// TIA Portal V17 export
// export: Created 2025-03-07T09:19:12.1414983Z, ExportSetting WithDefaults, DisplayName Totally Integrated Automation Portal, DisplayVersion V17 Update 8, DisplayName TIA Portal Openness, DisplayVersion V17 Update 8, DisplayName TIA Portal Version Control Interface, DisplayVersion V17, DisplayName SINAMICS Startdrive Advanced, DisplayVersion V17 SP2, DisplayName SINAMICS Startdrive G110M, G120, G120C, G120D, G120P, G115D, DisplayVersion V17 SP2, DisplayName SINAMICS Startdrive G130, G150, S120, S150, SINAMICS MV, S210, DisplayVersion V17 SP2, DisplayName STEP 7 Professional, DisplayVersion V17 Update 8, DisplayName SINUMERIK ONE STEP 7 Toolbox, DisplayVersion V17 Update 12, DisplayName SINUMERIK 840D sl STEP 7 Toolbox, DisplayVersion V17 Update 12, DisplayName STEP 7 Safety, DisplayVersion V17 Update 6, DisplayName WinCC Advanced, DisplayVersion V17 Update 8
FUNCTION "FC7225_HMI_AXES_CLADDING" : Void   // FC7225, LAD
{ S7_Optimized_Access := 'FALSE' }
AUTHOR : ETXETAR
VERSION : 1.0
// stored: AutoNumber false, IsIECCheckEnabled false, SetENOAutomatically false, UDAEnableTagReadback false
   VAR_TEMP
      ZERO : Byte;
      SOFTKEY_SELECT_PLUS : Byte;   // SOFTKEY_SELECT_PLUS
      SOFTKEY_SELECT_MINUS : Byte;   // SOFTKEY_SELECT_MINUS
      AXIS_SCREEN_SELECTED : Bool;   // AXIS SCREEN SELECTED
      SELECTED_AXIS : Int;   // SELECTED AXIS
   END_VAR
   VAR_TEMP   // added for the SCL form of the ladder/FBD networks
      _w1 : Bool;
      _w2 : Bool;
      _w3 : Bool;
      _w4 : Bool;
   END_VAR
BEGIN

REGION Network 1: ZERO
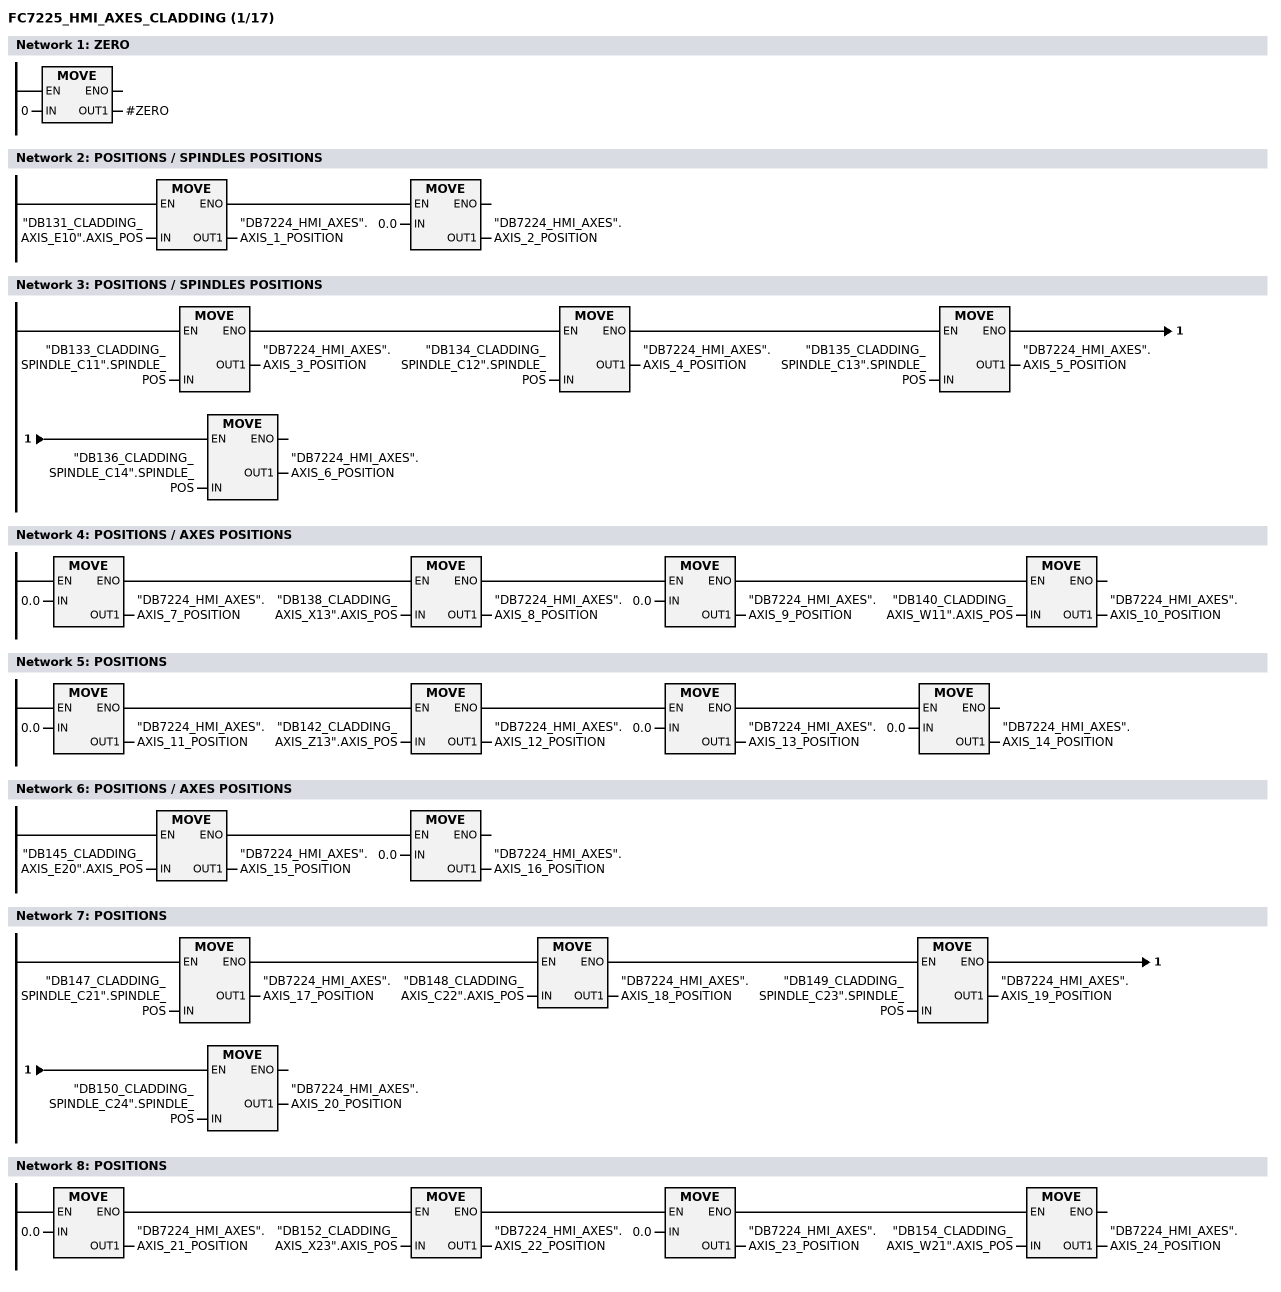
   RUNG wire#powerrail
      { S7_GenerateENO := "TRUE" } Move(in := 0, out1 => #ZERO)
   END_RUNG
   // the same network as SCL:
   #ZERO := 0;
END_REGION

REGION Network 2: POSITIONS / SPINDLES POSITIONS
   RUNG wire#powerrail
      { S7_GenerateENO := "TRUE" } Move(in := "DB131_CLADDING_AXIS_E10".AXIS_POS, out1 => "DB7224_HMI_AXES".AXIS_1_POSITION)
      { S7_GenerateENO := "TRUE" } Move(in := 0.0, out1 => "DB7224_HMI_AXES".AXIS_2_POSITION)
   END_RUNG
   // the same network as SCL:
   // ENO of a box is taken as its EN; it also drops when the box reports an error
   "DB7224_HMI_AXES".AXIS_1_POSITION := "DB131_CLADDING_AXIS_E10".AXIS_POS;
   "DB7224_HMI_AXES".AXIS_2_POSITION := 0.0;
END_REGION

REGION Network 3: POSITIONS / SPINDLES POSITIONS
   RUNG wire#powerrail
      { S7_GenerateENO := "TRUE" } Move(in := "DB133_CLADDING_SPINDLE_C11".SPINDLE_POS, out1 => "DB7224_HMI_AXES".AXIS_3_POSITION)
      { S7_GenerateENO := "TRUE" } Move(in := "DB134_CLADDING_SPINDLE_C12".SPINDLE_POS, out1 => "DB7224_HMI_AXES".AXIS_4_POSITION)
      { S7_GenerateENO := "TRUE" } Move(in := "DB135_CLADDING_SPINDLE_C13".SPINDLE_POS, out1 => "DB7224_HMI_AXES".AXIS_5_POSITION)
      { S7_GenerateENO := "TRUE" } Move(in := "DB136_CLADDING_SPINDLE_C14".SPINDLE_POS, out1 => "DB7224_HMI_AXES".AXIS_6_POSITION)
   END_RUNG
   // the same network as SCL:
   // ENO of a box is taken as its EN; it also drops when the box reports an error
   "DB7224_HMI_AXES".AXIS_3_POSITION := "DB133_CLADDING_SPINDLE_C11".SPINDLE_POS;
   "DB7224_HMI_AXES".AXIS_4_POSITION := "DB134_CLADDING_SPINDLE_C12".SPINDLE_POS;
   "DB7224_HMI_AXES".AXIS_5_POSITION := "DB135_CLADDING_SPINDLE_C13".SPINDLE_POS;
   "DB7224_HMI_AXES".AXIS_6_POSITION := "DB136_CLADDING_SPINDLE_C14".SPINDLE_POS;
END_REGION

REGION Network 4: POSITIONS / AXES POSITIONS
   RUNG wire#powerrail
      { S7_GenerateENO := "TRUE" } Move(in := 0.0, out1 => "DB7224_HMI_AXES".AXIS_7_POSITION)
      { S7_GenerateENO := "TRUE" } Move(in := "DB138_CLADDING_AXIS_X13".AXIS_POS, out1 => "DB7224_HMI_AXES".AXIS_8_POSITION)
      { S7_GenerateENO := "TRUE" } Move(in := 0.0, out1 => "DB7224_HMI_AXES".AXIS_9_POSITION)
      { S7_GenerateENO := "TRUE" } Move(in := "DB140_CLADDING_AXIS_W11".AXIS_POS, out1 => "DB7224_HMI_AXES".AXIS_10_POSITION)
   END_RUNG
   // the same network as SCL:
   // ENO of a box is taken as its EN; it also drops when the box reports an error
   "DB7224_HMI_AXES".AXIS_7_POSITION := 0.0;
   "DB7224_HMI_AXES".AXIS_8_POSITION := "DB138_CLADDING_AXIS_X13".AXIS_POS;
   "DB7224_HMI_AXES".AXIS_9_POSITION := 0.0;
   "DB7224_HMI_AXES".AXIS_10_POSITION := "DB140_CLADDING_AXIS_W11".AXIS_POS;
END_REGION

REGION Network 5: POSITIONS
   RUNG wire#powerrail
      { S7_GenerateENO := "TRUE" } Move(in := 0.0, out1 => "DB7224_HMI_AXES".AXIS_11_POSITION)
      { S7_GenerateENO := "TRUE" } Move(in := "DB142_CLADDING_AXIS_Z13".AXIS_POS, out1 => "DB7224_HMI_AXES".AXIS_12_POSITION)
      { S7_GenerateENO := "TRUE" } Move(in := 0.0, out1 => "DB7224_HMI_AXES".AXIS_13_POSITION)
      { S7_GenerateENO := "TRUE" } Move(in := 0.0, out1 => "DB7224_HMI_AXES".AXIS_14_POSITION)
   END_RUNG
   // the same network as SCL:
   // ENO of a box is taken as its EN; it also drops when the box reports an error
   "DB7224_HMI_AXES".AXIS_11_POSITION := 0.0;
   "DB7224_HMI_AXES".AXIS_12_POSITION := "DB142_CLADDING_AXIS_Z13".AXIS_POS;
   "DB7224_HMI_AXES".AXIS_13_POSITION := 0.0;
   "DB7224_HMI_AXES".AXIS_14_POSITION := 0.0;
END_REGION

REGION Network 6: POSITIONS / AXES POSITIONS
   RUNG wire#powerrail
      { S7_GenerateENO := "TRUE" } Move(in := "DB145_CLADDING_AXIS_E20".AXIS_POS, out1 => "DB7224_HMI_AXES".AXIS_15_POSITION)
      { S7_GenerateENO := "TRUE" } Move(in := 0.0, out1 => "DB7224_HMI_AXES".AXIS_16_POSITION)
   END_RUNG
   // the same network as SCL:
   // ENO of a box is taken as its EN; it also drops when the box reports an error
   "DB7224_HMI_AXES".AXIS_15_POSITION := "DB145_CLADDING_AXIS_E20".AXIS_POS;
   "DB7224_HMI_AXES".AXIS_16_POSITION := 0.0;
END_REGION

REGION Network 7: POSITIONS
   RUNG wire#powerrail
      { S7_GenerateENO := "TRUE" } Move(in := "DB147_CLADDING_SPINDLE_C21".SPINDLE_POS, out1 => "DB7224_HMI_AXES".AXIS_17_POSITION)
      { S7_GenerateENO := "TRUE" } Move(in := "DB148_CLADDING_AXIS_C22".AXIS_POS, out1 => "DB7224_HMI_AXES".AXIS_18_POSITION)
      { S7_GenerateENO := "TRUE" } Move(in := "DB149_CLADDING_SPINDLE_C23".SPINDLE_POS, out1 => "DB7224_HMI_AXES".AXIS_19_POSITION)
      { S7_GenerateENO := "TRUE" } Move(in := "DB150_CLADDING_SPINDLE_C24".SPINDLE_POS, out1 => "DB7224_HMI_AXES".AXIS_20_POSITION)
   END_RUNG
   // the same network as SCL:
   // ENO of a box is taken as its EN; it also drops when the box reports an error
   "DB7224_HMI_AXES".AXIS_17_POSITION := "DB147_CLADDING_SPINDLE_C21".SPINDLE_POS;
   "DB7224_HMI_AXES".AXIS_18_POSITION := "DB148_CLADDING_AXIS_C22".AXIS_POS;
   "DB7224_HMI_AXES".AXIS_19_POSITION := "DB149_CLADDING_SPINDLE_C23".SPINDLE_POS;
   "DB7224_HMI_AXES".AXIS_20_POSITION := "DB150_CLADDING_SPINDLE_C24".SPINDLE_POS;
END_REGION

REGION Network 8: POSITIONS
   RUNG wire#powerrail
      { S7_GenerateENO := "TRUE" } Move(in := 0.0, out1 => "DB7224_HMI_AXES".AXIS_21_POSITION)
      { S7_GenerateENO := "TRUE" } Move(in := "DB152_CLADDING_AXIS_X23".AXIS_POS, out1 => "DB7224_HMI_AXES".AXIS_22_POSITION)
      { S7_GenerateENO := "TRUE" } Move(in := 0.0, out1 => "DB7224_HMI_AXES".AXIS_23_POSITION)
      { S7_GenerateENO := "TRUE" } Move(in := "DB154_CLADDING_AXIS_W21".AXIS_POS, out1 => "DB7224_HMI_AXES".AXIS_24_POSITION)
   END_RUNG
   // the same network as SCL:
   // ENO of a box is taken as its EN; it also drops when the box reports an error
   "DB7224_HMI_AXES".AXIS_21_POSITION := 0.0;
   "DB7224_HMI_AXES".AXIS_22_POSITION := "DB152_CLADDING_AXIS_X23".AXIS_POS;
   "DB7224_HMI_AXES".AXIS_23_POSITION := 0.0;
   "DB7224_HMI_AXES".AXIS_24_POSITION := "DB154_CLADDING_AXIS_W21".AXIS_POS;
END_REGION

REGION Network 9: POSITIONS
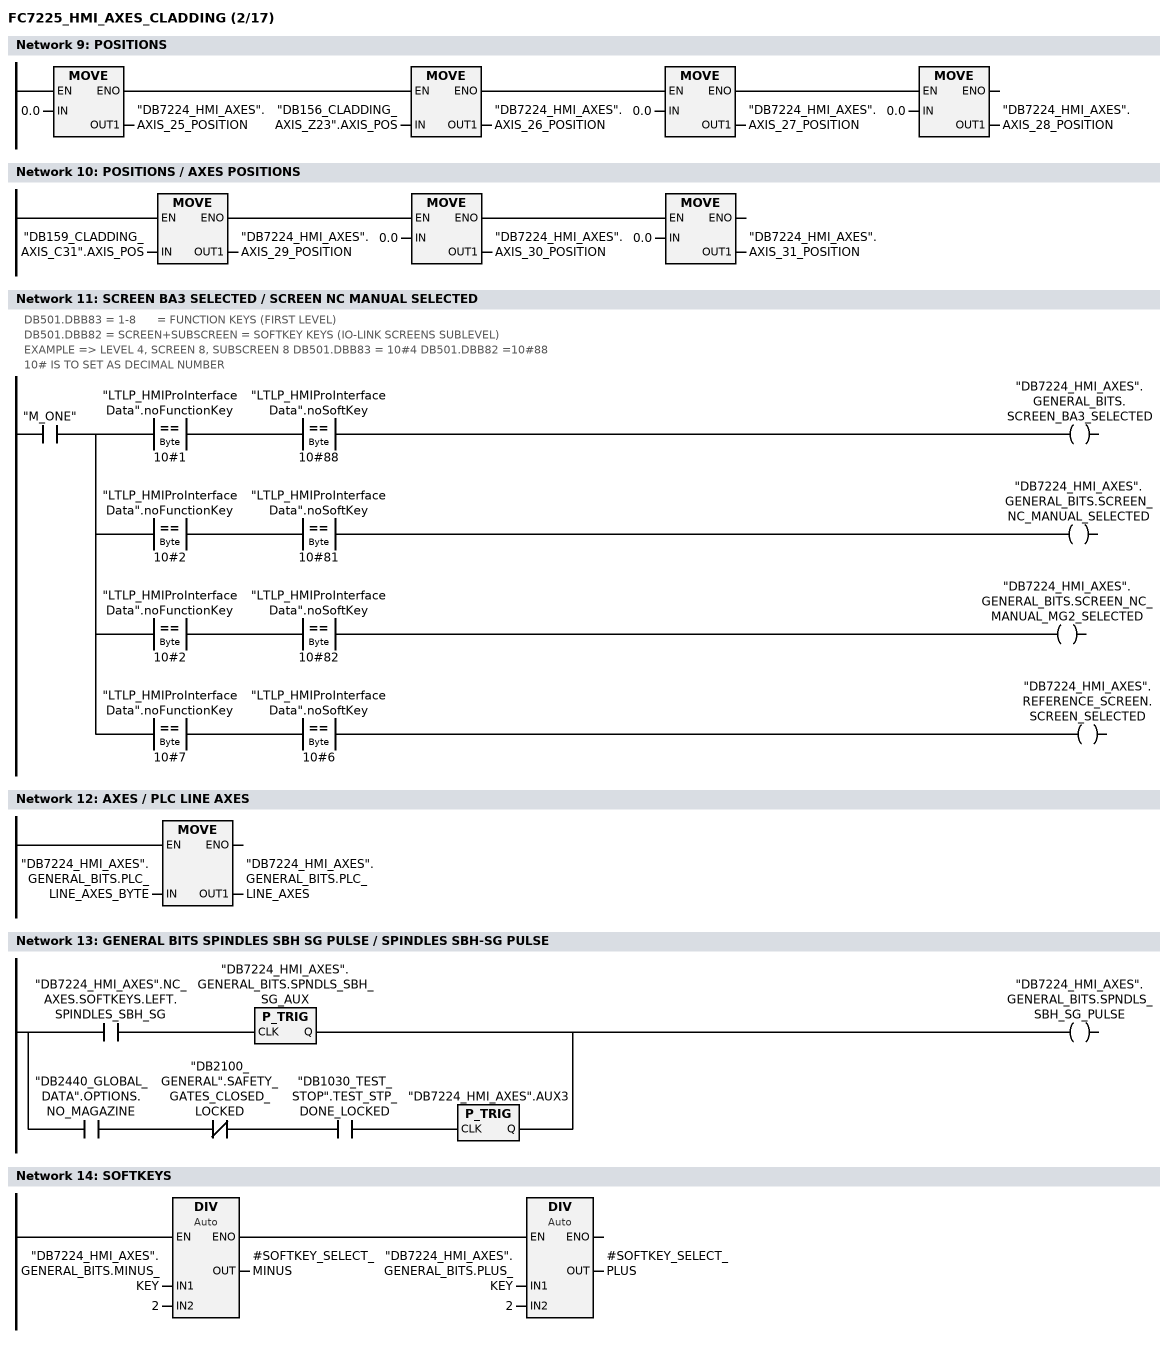
   RUNG wire#powerrail
      { S7_GenerateENO := "TRUE" } Move(in := 0.0, out1 => "DB7224_HMI_AXES".AXIS_25_POSITION)
      { S7_GenerateENO := "TRUE" } Move(in := "DB156_CLADDING_AXIS_Z23".AXIS_POS, out1 => "DB7224_HMI_AXES".AXIS_26_POSITION)
      { S7_GenerateENO := "TRUE" } Move(in := 0.0, out1 => "DB7224_HMI_AXES".AXIS_27_POSITION)
      { S7_GenerateENO := "TRUE" } Move(in := 0.0, out1 => "DB7224_HMI_AXES".AXIS_28_POSITION)
   END_RUNG
   // the same network as SCL:
   // ENO of a box is taken as its EN; it also drops when the box reports an error
   "DB7224_HMI_AXES".AXIS_25_POSITION := 0.0;
   "DB7224_HMI_AXES".AXIS_26_POSITION := "DB156_CLADDING_AXIS_Z23".AXIS_POS;
   "DB7224_HMI_AXES".AXIS_27_POSITION := 0.0;
   "DB7224_HMI_AXES".AXIS_28_POSITION := 0.0;
END_REGION

REGION Network 10: POSITIONS / AXES POSITIONS
   RUNG wire#powerrail
      { S7_GenerateENO := "TRUE" } Move(in := "DB159_CLADDING_AXIS_C31".AXIS_POS, out1 => "DB7224_HMI_AXES".AXIS_29_POSITION)
      { S7_GenerateENO := "TRUE" } Move(in := 0.0, out1 => "DB7224_HMI_AXES".AXIS_30_POSITION)
      { S7_GenerateENO := "TRUE" } Move(in := 0.0, out1 => "DB7224_HMI_AXES".AXIS_31_POSITION)
   END_RUNG
   // the same network as SCL:
   // ENO of a box is taken as its EN; it also drops when the box reports an error
   "DB7224_HMI_AXES".AXIS_29_POSITION := "DB159_CLADDING_AXIS_C31".AXIS_POS;
   "DB7224_HMI_AXES".AXIS_30_POSITION := 0.0;
   "DB7224_HMI_AXES".AXIS_31_POSITION := 0.0;
END_REGION

REGION Network 11: SCREEN BA3 SELECTED / SCREEN NC MANUAL SELECTED
   // DB501.DBB83 = 1-8      = FUNCTION KEYS (FIRST LEVEL)
   // DB501.DBB82 = SCREEN+SUBSCREEN = SOFTKEY KEYS (IO-LINK SCREENS SUBLEVEL)
   // EXAMPLE => LEVEL 4, SCREEN 8, SUBSCREEN 8 DB501.DBB83 = 10#4 DB501.DBB82 =10#88
   // 10# IS TO SET AS DECIMAL NUMBER
   RUNG wire#powerrail
      Contact( "M_ONE" )
      wire#w1
      { S7_Templates := "SrcType := Byte" } EQ_Contact(in1 := "LTLP_HMIProInterfaceData".noFunctionKey, in2 := 10#1)
      { S7_Templates := "SrcType := Byte" } EQ_Contact(in1 := "LTLP_HMIProInterfaceData".noSoftKey, in2 := 10#88)
      Coil( "DB7224_HMI_AXES".GENERAL_BITS.SCREEN_BA3_SELECTED )
   END_RUNG
   RUNG wire#w1
      { S7_Templates := "SrcType := Byte" } EQ_Contact(in1 := "LTLP_HMIProInterfaceData".noFunctionKey, in2 := 10#2)
      { S7_Templates := "SrcType := Byte" } EQ_Contact(in1 := "LTLP_HMIProInterfaceData".noSoftKey, in2 := 10#81)
      Coil( "DB7224_HMI_AXES".GENERAL_BITS.SCREEN_NC_MANUAL_SELECTED )
   END_RUNG
   RUNG wire#w1
      { S7_Templates := "SrcType := Byte" } EQ_Contact(in1 := "LTLP_HMIProInterfaceData".noFunctionKey, in2 := 10#2)
      { S7_Templates := "SrcType := Byte" } EQ_Contact(in1 := "LTLP_HMIProInterfaceData".noSoftKey, in2 := 10#82)
      Coil( "DB7224_HMI_AXES".GENERAL_BITS.SCREEN_NC_MANUAL_MG2_SELECTED )
   END_RUNG
   RUNG wire#w1
      { S7_Templates := "SrcType := Byte" } EQ_Contact(in1 := "LTLP_HMIProInterfaceData".noFunctionKey, in2 := 10#7)
      { S7_Templates := "SrcType := Byte" } EQ_Contact(in1 := "LTLP_HMIProInterfaceData".noSoftKey, in2 := 10#6)
      Coil( "DB7224_HMI_AXES".REFERENCE_SCREEN.SCREEN_SELECTED )
   END_RUNG
   // the same network as SCL:
   "DB7224_HMI_AXES".GENERAL_BITS.SCREEN_BA3_SELECTED := "M_ONE" AND ("LTLP_HMIProInterfaceData".noFunctionKey = 10#1) AND ("LTLP_HMIProInterfaceData".noSoftKey = 10#88);
   "DB7224_HMI_AXES".GENERAL_BITS.SCREEN_NC_MANUAL_SELECTED := "M_ONE" AND ("LTLP_HMIProInterfaceData".noFunctionKey = 10#2) AND ("LTLP_HMIProInterfaceData".noSoftKey = 10#81);
   "DB7224_HMI_AXES".GENERAL_BITS.SCREEN_NC_MANUAL_MG2_SELECTED := "M_ONE" AND ("LTLP_HMIProInterfaceData".noFunctionKey = 10#2) AND ("LTLP_HMIProInterfaceData".noSoftKey = 10#82);
   "DB7224_HMI_AXES".REFERENCE_SCREEN.SCREEN_SELECTED := "M_ONE" AND ("LTLP_HMIProInterfaceData".noFunctionKey = 10#7) AND ("LTLP_HMIProInterfaceData".noSoftKey = 10#6);
END_REGION

REGION Network 12: AXES / PLC LINE AXES
   RUNG wire#powerrail
      { S7_GenerateENO := "TRUE" } Move(in := "DB7224_HMI_AXES".GENERAL_BITS.PLC_LINE_AXES_BYTE, out1 => "DB7224_HMI_AXES".GENERAL_BITS.PLC_LINE_AXES)
   END_RUNG
   // the same network as SCL:
   "DB7224_HMI_AXES".GENERAL_BITS.PLC_LINE_AXES := "DB7224_HMI_AXES".GENERAL_BITS.PLC_LINE_AXES_BYTE;
END_REGION

REGION Network 13: GENERAL BITS SPINDLES SBH SG PULSE / SPINDLES SBH-SG PULSE
   RUNG wire#powerrail
      Contact( "DB7224_HMI_AXES".NC_AXES.SOFTKEYS.LEFT.SPINDLES_SBH_SG )
      P_Trig( "DB7224_HMI_AXES".GENERAL_BITS.SPNDLS_SBH_SG_AUX )
      wire#w1
      Coil( "DB7224_HMI_AXES".GENERAL_BITS.SPNDLS_SBH_SG_PULSE )
   END_RUNG
   RUNG wire#powerrail
      Contact( "DB2440_GLOBAL_DATA".OPTIONS.NO_MAGAZINE )
      I_Contact( "DB2100_GENERAL".SAFETY_GATES_CLOSED_LOCKED )
      Contact( "DB1030_TEST_STOP".TEST_STP_DONE_LOCKED )
      P_Trig( "DB7224_HMI_AXES".AUX3 )
   END_RUNG wire#w1
   // the same network as SCL:
   #_w1 := "DB7224_HMI_AXES".NC_AXES.SOFTKEYS.LEFT.SPINDLES_SBH_SG AND NOT "DB7224_HMI_AXES".GENERAL_BITS.SPNDLS_SBH_SG_AUX;   // rising edge
   "DB7224_HMI_AXES".GENERAL_BITS.SPNDLS_SBH_SG_AUX := "DB7224_HMI_AXES".NC_AXES.SOFTKEYS.LEFT.SPINDLES_SBH_SG;
   #_w2 := "DB2440_GLOBAL_DATA".OPTIONS.NO_MAGAZINE AND NOT "DB2100_GENERAL".SAFETY_GATES_CLOSED_LOCKED AND "DB1030_TEST_STOP".TEST_STP_DONE_LOCKED;
   #_w3 := #_w2 AND NOT "DB7224_HMI_AXES".AUX3;   // rising edge
   "DB7224_HMI_AXES".AUX3 := #_w2;
   "DB7224_HMI_AXES".GENERAL_BITS.SPNDLS_SBH_SG_PULSE := #_w1 OR #_w3;
END_REGION

REGION Network 14: SOFTKEYS
   RUNG wire#powerrail
      Div(in1 := "DB7224_HMI_AXES".GENERAL_BITS.MINUS_KEY, in2 := 2, out => #SOFTKEY_SELECT_MINUS)
      Div(in1 := "DB7224_HMI_AXES".GENERAL_BITS.PLUS_KEY, in2 := 2, out => #SOFTKEY_SELECT_PLUS)
   END_RUNG
   // the same network as SCL:
   #SOFTKEY_SELECT_MINUS := "DB7224_HMI_AXES".GENERAL_BITS.MINUS_KEY / 2;
   #SOFTKEY_SELECT_PLUS := "DB7224_HMI_AXES".GENERAL_BITS.PLUS_KEY / 2;
END_REGION

REGION Network 15: SOFTKEYS / LEFT MINUS SOFTKEYS
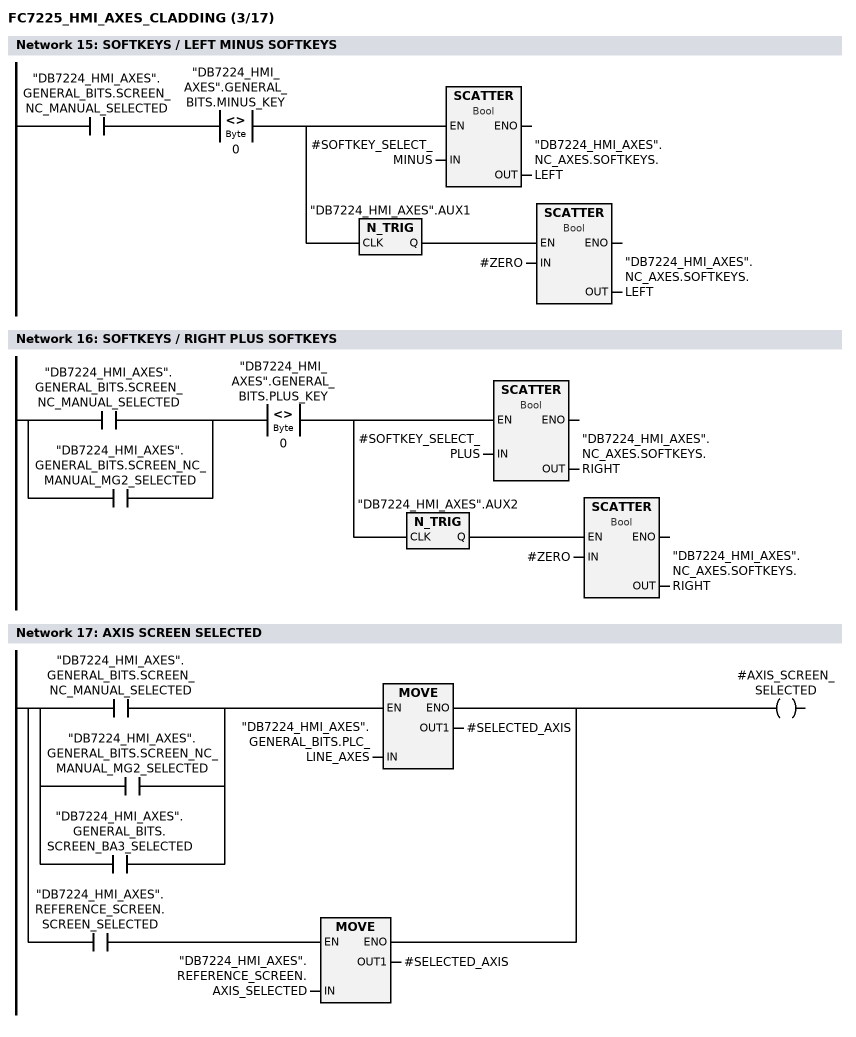
   RUNG wire#powerrail
      Contact( "DB7224_HMI_AXES".GENERAL_BITS.SCREEN_NC_MANUAL_SELECTED )
      { S7_Templates := "SrcType := Byte" } NE_Contact(in1 := "DB7224_HMI_AXES".GENERAL_BITS.MINUS_KEY, in2 := 0)
      wire#w1
      { S7_Templates := "[dest_type := Bool, src_type := Byte]" } SCATTER(IN := #SOFTKEY_SELECT_MINUS, OUT => "DB7224_HMI_AXES".NC_AXES.SOFTKEYS.LEFT)
   END_RUNG
   RUNG wire#w1
      N_Trig( "DB7224_HMI_AXES".AUX1 )
      { S7_Templates := "[dest_type := Bool, src_type := Byte]" } SCATTER(IN := #ZERO, OUT => "DB7224_HMI_AXES".NC_AXES.SOFTKEYS.LEFT)
   END_RUNG
   // the same network as SCL:
   #_w1 := "DB7224_HMI_AXES".GENERAL_BITS.SCREEN_NC_MANUAL_SELECTED AND ("DB7224_HMI_AXES".GENERAL_BITS.MINUS_KEY <> 0);
   IF #_w1 THEN SCATTER(IN := #SOFTKEY_SELECT_MINUS, OUT => "DB7224_HMI_AXES".NC_AXES.SOFTKEYS.LEFT); END_IF;
   #_w2 := NOT #_w1 AND "DB7224_HMI_AXES".AUX1;   // falling edge
   "DB7224_HMI_AXES".AUX1 := #_w1;
   IF #_w2 THEN SCATTER(IN := #ZERO, OUT => "DB7224_HMI_AXES".NC_AXES.SOFTKEYS.LEFT); END_IF;
END_REGION

REGION Network 16: SOFTKEYS / RIGHT PLUS SOFTKEYS
   RUNG wire#powerrail
      Contact( "DB7224_HMI_AXES".GENERAL_BITS.SCREEN_NC_MANUAL_SELECTED )
      wire#w1
      { S7_Templates := "SrcType := Byte" } NE_Contact(in1 := "DB7224_HMI_AXES".GENERAL_BITS.PLUS_KEY, in2 := 0)
      wire#w2
      { S7_Templates := "[dest_type := Bool, src_type := Byte]" } SCATTER(IN := #SOFTKEY_SELECT_PLUS, OUT => "DB7224_HMI_AXES".NC_AXES.SOFTKEYS.RIGHT)
   END_RUNG
   RUNG wire#powerrail
      Contact( "DB7224_HMI_AXES".GENERAL_BITS.SCREEN_NC_MANUAL_MG2_SELECTED )
   END_RUNG wire#w1
   RUNG wire#w2
      N_Trig( "DB7224_HMI_AXES".AUX2 )
      { S7_Templates := "[dest_type := Bool, src_type := Byte]" } SCATTER(IN := #ZERO, OUT => "DB7224_HMI_AXES".NC_AXES.SOFTKEYS.RIGHT)
   END_RUNG
   // the same network as SCL:
   #_w1 := ("DB7224_HMI_AXES".GENERAL_BITS.SCREEN_NC_MANUAL_SELECTED OR "DB7224_HMI_AXES".GENERAL_BITS.SCREEN_NC_MANUAL_MG2_SELECTED) AND ("DB7224_HMI_AXES".GENERAL_BITS.PLUS_KEY <> 0);
   IF #_w1 THEN SCATTER(IN := #SOFTKEY_SELECT_PLUS, OUT => "DB7224_HMI_AXES".NC_AXES.SOFTKEYS.RIGHT); END_IF;
   #_w2 := NOT #_w1 AND "DB7224_HMI_AXES".AUX2;   // falling edge
   "DB7224_HMI_AXES".AUX2 := #_w1;
   IF #_w2 THEN SCATTER(IN := #ZERO, OUT => "DB7224_HMI_AXES".NC_AXES.SOFTKEYS.RIGHT); END_IF;
END_REGION

REGION Network 17: AXIS SCREEN SELECTED
   RUNG wire#powerrail
      Contact( "DB7224_HMI_AXES".GENERAL_BITS.SCREEN_NC_MANUAL_SELECTED )
      wire#w1
      Move(in := "DB7224_HMI_AXES".GENERAL_BITS.PLC_LINE_AXES, out1 => #SELECTED_AXIS)
      wire#w2
      Coil( #AXIS_SCREEN_SELECTED )
   END_RUNG
   RUNG wire#powerrail
      Contact( "DB7224_HMI_AXES".GENERAL_BITS.SCREEN_NC_MANUAL_MG2_SELECTED )
   END_RUNG wire#w1
   RUNG wire#powerrail
      Contact( "DB7224_HMI_AXES".GENERAL_BITS.SCREEN_BA3_SELECTED )
   END_RUNG wire#w1
   RUNG wire#powerrail
      Contact( "DB7224_HMI_AXES".REFERENCE_SCREEN.SCREEN_SELECTED )
      Move(in := "DB7224_HMI_AXES".REFERENCE_SCREEN.AXIS_SELECTED, out1 => #SELECTED_AXIS)
   END_RUNG wire#w2
   // the same network as SCL:
   #_w1 := "DB7224_HMI_AXES".GENERAL_BITS.SCREEN_NC_MANUAL_SELECTED OR "DB7224_HMI_AXES".GENERAL_BITS.SCREEN_NC_MANUAL_MG2_SELECTED OR "DB7224_HMI_AXES".GENERAL_BITS.SCREEN_BA3_SELECTED;
   IF #_w1 THEN #SELECTED_AXIS := "DB7224_HMI_AXES".GENERAL_BITS.PLC_LINE_AXES; END_IF;
   IF "DB7224_HMI_AXES".REFERENCE_SCREEN.SCREEN_SELECTED THEN
       #SELECTED_AXIS := "DB7224_HMI_AXES".REFERENCE_SCREEN.AXIS_SELECTED;
   END_IF;
   #AXIS_SCREEN_SELECTED := #_w1 OR "DB7224_HMI_AXES".REFERENCE_SCREEN.SCREEN_SELECTED;
END_REGION

REGION Network 18: AXES SELECTED / SPINDLES SELECTED
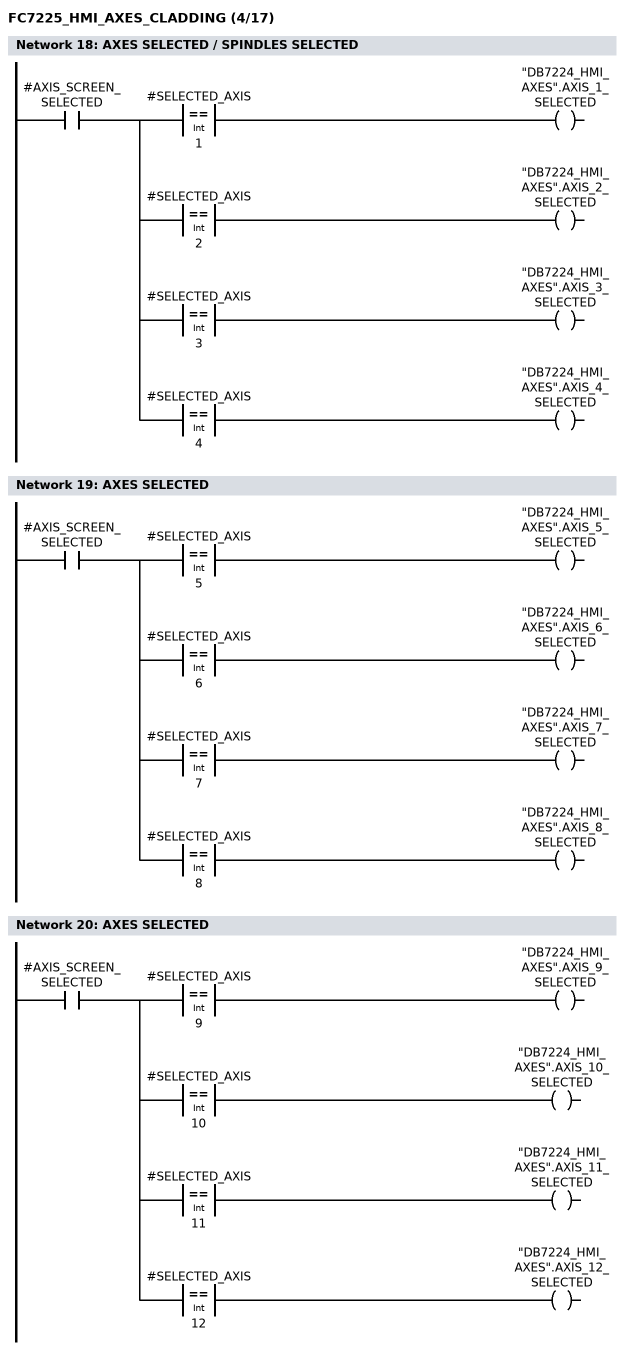
   RUNG wire#powerrail
      Contact( #AXIS_SCREEN_SELECTED )
      wire#w1
      { S7_Templates := "SrcType := Int" } EQ_Contact(in1 := #SELECTED_AXIS, in2 := 1)
      Coil( "DB7224_HMI_AXES".AXIS_1_SELECTED )
   END_RUNG
   RUNG wire#w1
      { S7_Templates := "SrcType := Int" } EQ_Contact(in1 := #SELECTED_AXIS, in2 := 2)
      Coil( "DB7224_HMI_AXES".AXIS_2_SELECTED )
   END_RUNG
   RUNG wire#w1
      { S7_Templates := "SrcType := Int" } EQ_Contact(in1 := #SELECTED_AXIS, in2 := 3)
      Coil( "DB7224_HMI_AXES".AXIS_3_SELECTED )
   END_RUNG
   RUNG wire#w1
      { S7_Templates := "SrcType := Int" } EQ_Contact(in1 := #SELECTED_AXIS, in2 := 4)
      Coil( "DB7224_HMI_AXES".AXIS_4_SELECTED )
   END_RUNG
   // the same network as SCL:
   "DB7224_HMI_AXES".AXIS_1_SELECTED := #AXIS_SCREEN_SELECTED AND (#SELECTED_AXIS = 1);
   "DB7224_HMI_AXES".AXIS_2_SELECTED := #AXIS_SCREEN_SELECTED AND (#SELECTED_AXIS = 2);
   "DB7224_HMI_AXES".AXIS_3_SELECTED := #AXIS_SCREEN_SELECTED AND (#SELECTED_AXIS = 3);
   "DB7224_HMI_AXES".AXIS_4_SELECTED := #AXIS_SCREEN_SELECTED AND (#SELECTED_AXIS = 4);
END_REGION

REGION Network 19: AXES SELECTED
   RUNG wire#powerrail
      Contact( #AXIS_SCREEN_SELECTED )
      wire#w1
      { S7_Templates := "SrcType := Int" } EQ_Contact(in1 := #SELECTED_AXIS, in2 := 5)
      Coil( "DB7224_HMI_AXES".AXIS_5_SELECTED )
   END_RUNG
   RUNG wire#w1
      { S7_Templates := "SrcType := Int" } EQ_Contact(in1 := #SELECTED_AXIS, in2 := 6)
      Coil( "DB7224_HMI_AXES".AXIS_6_SELECTED )
   END_RUNG
   RUNG wire#w1
      { S7_Templates := "SrcType := Int" } EQ_Contact(in1 := #SELECTED_AXIS, in2 := 7)
      Coil( "DB7224_HMI_AXES".AXIS_7_SELECTED )
   END_RUNG
   RUNG wire#w1
      { S7_Templates := "SrcType := Int" } EQ_Contact(in1 := #SELECTED_AXIS, in2 := 8)
      Coil( "DB7224_HMI_AXES".AXIS_8_SELECTED )
   END_RUNG
   // the same network as SCL:
   "DB7224_HMI_AXES".AXIS_5_SELECTED := #AXIS_SCREEN_SELECTED AND (#SELECTED_AXIS = 5);
   "DB7224_HMI_AXES".AXIS_6_SELECTED := #AXIS_SCREEN_SELECTED AND (#SELECTED_AXIS = 6);
   "DB7224_HMI_AXES".AXIS_7_SELECTED := #AXIS_SCREEN_SELECTED AND (#SELECTED_AXIS = 7);
   "DB7224_HMI_AXES".AXIS_8_SELECTED := #AXIS_SCREEN_SELECTED AND (#SELECTED_AXIS = 8);
END_REGION

REGION Network 20: AXES SELECTED
   RUNG wire#powerrail
      Contact( #AXIS_SCREEN_SELECTED )
      wire#w1
      { S7_Templates := "SrcType := Int" } EQ_Contact(in1 := #SELECTED_AXIS, in2 := 9)
      Coil( "DB7224_HMI_AXES".AXIS_9_SELECTED )
   END_RUNG
   RUNG wire#w1
      { S7_Templates := "SrcType := Int" } EQ_Contact(in1 := #SELECTED_AXIS, in2 := 10)
      Coil( "DB7224_HMI_AXES".AXIS_10_SELECTED )
   END_RUNG
   RUNG wire#w1
      { S7_Templates := "SrcType := Int" } EQ_Contact(in1 := #SELECTED_AXIS, in2 := 11)
      Coil( "DB7224_HMI_AXES".AXIS_11_SELECTED )
   END_RUNG
   RUNG wire#w1
      { S7_Templates := "SrcType := Int" } EQ_Contact(in1 := #SELECTED_AXIS, in2 := 12)
      Coil( "DB7224_HMI_AXES".AXIS_12_SELECTED )
   END_RUNG
   // the same network as SCL:
   "DB7224_HMI_AXES".AXIS_9_SELECTED := #AXIS_SCREEN_SELECTED AND (#SELECTED_AXIS = 9);
   "DB7224_HMI_AXES".AXIS_10_SELECTED := #AXIS_SCREEN_SELECTED AND (#SELECTED_AXIS = 10);
   "DB7224_HMI_AXES".AXIS_11_SELECTED := #AXIS_SCREEN_SELECTED AND (#SELECTED_AXIS = 11);
   "DB7224_HMI_AXES".AXIS_12_SELECTED := #AXIS_SCREEN_SELECTED AND (#SELECTED_AXIS = 12);
END_REGION

REGION Network 21: AXES SELECTED
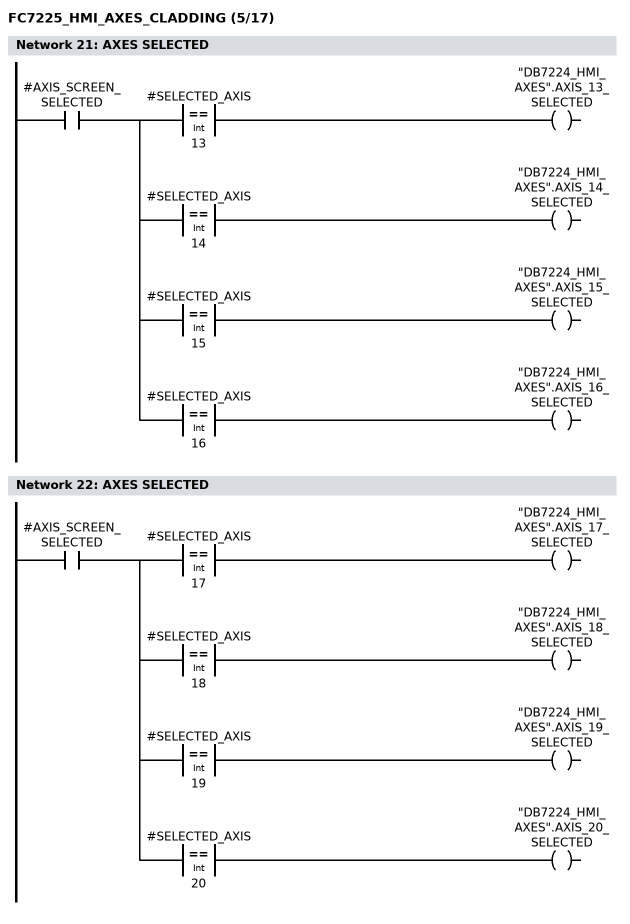
   RUNG wire#powerrail
      Contact( #AXIS_SCREEN_SELECTED )
      wire#w1
      { S7_Templates := "SrcType := Int" } EQ_Contact(in1 := #SELECTED_AXIS, in2 := 13)
      Coil( "DB7224_HMI_AXES".AXIS_13_SELECTED )
   END_RUNG
   RUNG wire#w1
      { S7_Templates := "SrcType := Int" } EQ_Contact(in1 := #SELECTED_AXIS, in2 := 14)
      Coil( "DB7224_HMI_AXES".AXIS_14_SELECTED )
   END_RUNG
   RUNG wire#w1
      { S7_Templates := "SrcType := Int" } EQ_Contact(in1 := #SELECTED_AXIS, in2 := 15)
      Coil( "DB7224_HMI_AXES".AXIS_15_SELECTED )
   END_RUNG
   RUNG wire#w1
      { S7_Templates := "SrcType := Int" } EQ_Contact(in1 := #SELECTED_AXIS, in2 := 16)
      Coil( "DB7224_HMI_AXES".AXIS_16_SELECTED )
   END_RUNG
   // the same network as SCL:
   "DB7224_HMI_AXES".AXIS_13_SELECTED := #AXIS_SCREEN_SELECTED AND (#SELECTED_AXIS = 13);
   "DB7224_HMI_AXES".AXIS_14_SELECTED := #AXIS_SCREEN_SELECTED AND (#SELECTED_AXIS = 14);
   "DB7224_HMI_AXES".AXIS_15_SELECTED := #AXIS_SCREEN_SELECTED AND (#SELECTED_AXIS = 15);
   "DB7224_HMI_AXES".AXIS_16_SELECTED := #AXIS_SCREEN_SELECTED AND (#SELECTED_AXIS = 16);
END_REGION

REGION Network 22: AXES SELECTED
   RUNG wire#powerrail
      Contact( #AXIS_SCREEN_SELECTED )
      wire#w1
      { S7_Templates := "SrcType := Int" } EQ_Contact(in1 := #SELECTED_AXIS, in2 := 17)
      Coil( "DB7224_HMI_AXES".AXIS_17_SELECTED )
   END_RUNG
   RUNG wire#w1
      { S7_Templates := "SrcType := Int" } EQ_Contact(in1 := #SELECTED_AXIS, in2 := 18)
      Coil( "DB7224_HMI_AXES".AXIS_18_SELECTED )
   END_RUNG
   RUNG wire#w1
      { S7_Templates := "SrcType := Int" } EQ_Contact(in1 := #SELECTED_AXIS, in2 := 19)
      Coil( "DB7224_HMI_AXES".AXIS_19_SELECTED )
   END_RUNG
   RUNG wire#w1
      { S7_Templates := "SrcType := Int" } EQ_Contact(in1 := #SELECTED_AXIS, in2 := 20)
      Coil( "DB7224_HMI_AXES".AXIS_20_SELECTED )
   END_RUNG
   // the same network as SCL:
   "DB7224_HMI_AXES".AXIS_17_SELECTED := #AXIS_SCREEN_SELECTED AND (#SELECTED_AXIS = 17);
   "DB7224_HMI_AXES".AXIS_18_SELECTED := #AXIS_SCREEN_SELECTED AND (#SELECTED_AXIS = 18);
   "DB7224_HMI_AXES".AXIS_19_SELECTED := #AXIS_SCREEN_SELECTED AND (#SELECTED_AXIS = 19);
   "DB7224_HMI_AXES".AXIS_20_SELECTED := #AXIS_SCREEN_SELECTED AND (#SELECTED_AXIS = 20);
END_REGION

REGION Network 23: AXES SELECTED
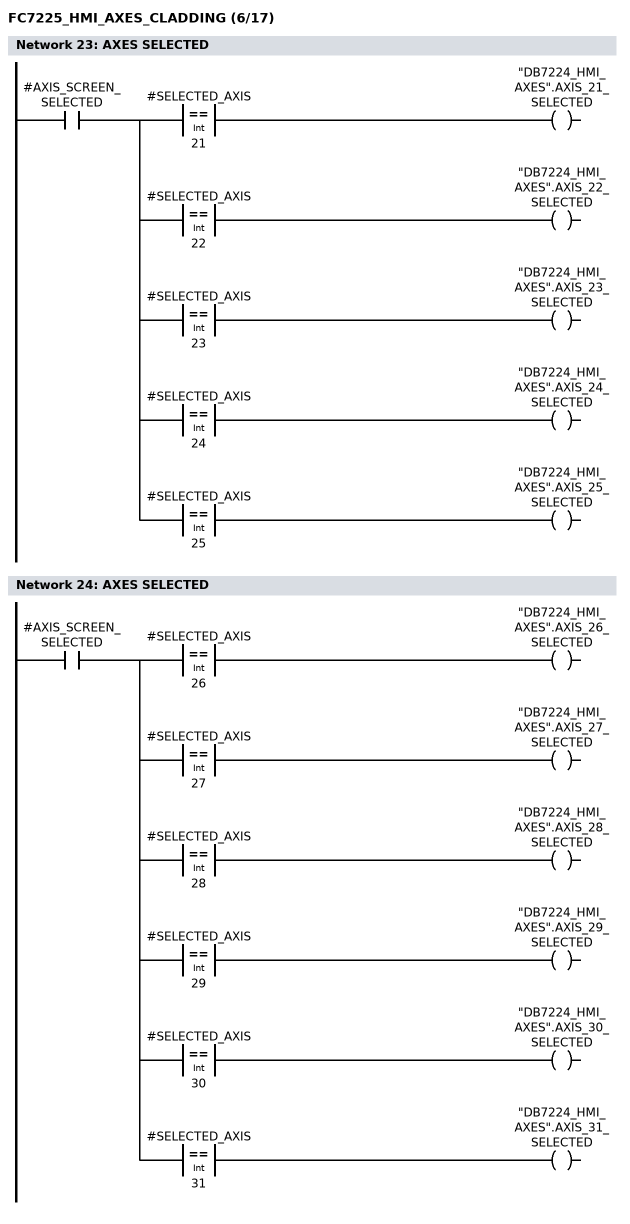
   RUNG wire#powerrail
      Contact( #AXIS_SCREEN_SELECTED )
      wire#w1
      { S7_Templates := "SrcType := Int" } EQ_Contact(in1 := #SELECTED_AXIS, in2 := 21)
      Coil( "DB7224_HMI_AXES".AXIS_21_SELECTED )
   END_RUNG
   RUNG wire#w1
      { S7_Templates := "SrcType := Int" } EQ_Contact(in1 := #SELECTED_AXIS, in2 := 22)
      Coil( "DB7224_HMI_AXES".AXIS_22_SELECTED )
   END_RUNG
   RUNG wire#w1
      { S7_Templates := "SrcType := Int" } EQ_Contact(in1 := #SELECTED_AXIS, in2 := 23)
      Coil( "DB7224_HMI_AXES".AXIS_23_SELECTED )
   END_RUNG
   RUNG wire#w1
      { S7_Templates := "SrcType := Int" } EQ_Contact(in1 := #SELECTED_AXIS, in2 := 24)
      Coil( "DB7224_HMI_AXES".AXIS_24_SELECTED )
   END_RUNG
   RUNG wire#w1
      { S7_Templates := "SrcType := Int" } EQ_Contact(in1 := #SELECTED_AXIS, in2 := 25)
      Coil( "DB7224_HMI_AXES".AXIS_25_SELECTED )
   END_RUNG
   // the same network as SCL:
   "DB7224_HMI_AXES".AXIS_21_SELECTED := #AXIS_SCREEN_SELECTED AND (#SELECTED_AXIS = 21);
   "DB7224_HMI_AXES".AXIS_22_SELECTED := #AXIS_SCREEN_SELECTED AND (#SELECTED_AXIS = 22);
   "DB7224_HMI_AXES".AXIS_23_SELECTED := #AXIS_SCREEN_SELECTED AND (#SELECTED_AXIS = 23);
   "DB7224_HMI_AXES".AXIS_24_SELECTED := #AXIS_SCREEN_SELECTED AND (#SELECTED_AXIS = 24);
   "DB7224_HMI_AXES".AXIS_25_SELECTED := #AXIS_SCREEN_SELECTED AND (#SELECTED_AXIS = 25);
END_REGION

REGION Network 24: AXES SELECTED
   RUNG wire#powerrail
      Contact( #AXIS_SCREEN_SELECTED )
      wire#w1
      { S7_Templates := "SrcType := Int" } EQ_Contact(in1 := #SELECTED_AXIS, in2 := 26)
      Coil( "DB7224_HMI_AXES".AXIS_26_SELECTED )
   END_RUNG
   RUNG wire#w1
      { S7_Templates := "SrcType := Int" } EQ_Contact(in1 := #SELECTED_AXIS, in2 := 27)
      Coil( "DB7224_HMI_AXES".AXIS_27_SELECTED )
   END_RUNG
   RUNG wire#w1
      { S7_Templates := "SrcType := Int" } EQ_Contact(in1 := #SELECTED_AXIS, in2 := 28)
      Coil( "DB7224_HMI_AXES".AXIS_28_SELECTED )
   END_RUNG
   RUNG wire#w1
      { S7_Templates := "SrcType := Int" } EQ_Contact(in1 := #SELECTED_AXIS, in2 := 29)
      Coil( "DB7224_HMI_AXES".AXIS_29_SELECTED )
   END_RUNG
   RUNG wire#w1
      { S7_Templates := "SrcType := Int" } EQ_Contact(in1 := #SELECTED_AXIS, in2 := 30)
      Coil( "DB7224_HMI_AXES".AXIS_30_SELECTED )
   END_RUNG
   RUNG wire#w1
      { S7_Templates := "SrcType := Int" } EQ_Contact(in1 := #SELECTED_AXIS, in2 := 31)
      Coil( "DB7224_HMI_AXES".AXIS_31_SELECTED )
   END_RUNG
   // the same network as SCL:
   "DB7224_HMI_AXES".AXIS_26_SELECTED := #AXIS_SCREEN_SELECTED AND (#SELECTED_AXIS = 26);
   "DB7224_HMI_AXES".AXIS_27_SELECTED := #AXIS_SCREEN_SELECTED AND (#SELECTED_AXIS = 27);
   "DB7224_HMI_AXES".AXIS_28_SELECTED := #AXIS_SCREEN_SELECTED AND (#SELECTED_AXIS = 28);
   "DB7224_HMI_AXES".AXIS_29_SELECTED := #AXIS_SCREEN_SELECTED AND (#SELECTED_AXIS = 29);
   "DB7224_HMI_AXES".AXIS_30_SELECTED := #AXIS_SCREEN_SELECTED AND (#SELECTED_AXIS = 30);
   "DB7224_HMI_AXES".AXIS_31_SELECTED := #AXIS_SCREEN_SELECTED AND (#SELECTED_AXIS = 31);
END_REGION

REGION Network 25: AXIS REFERENCED / SPINDLES/AXES REFERENCED
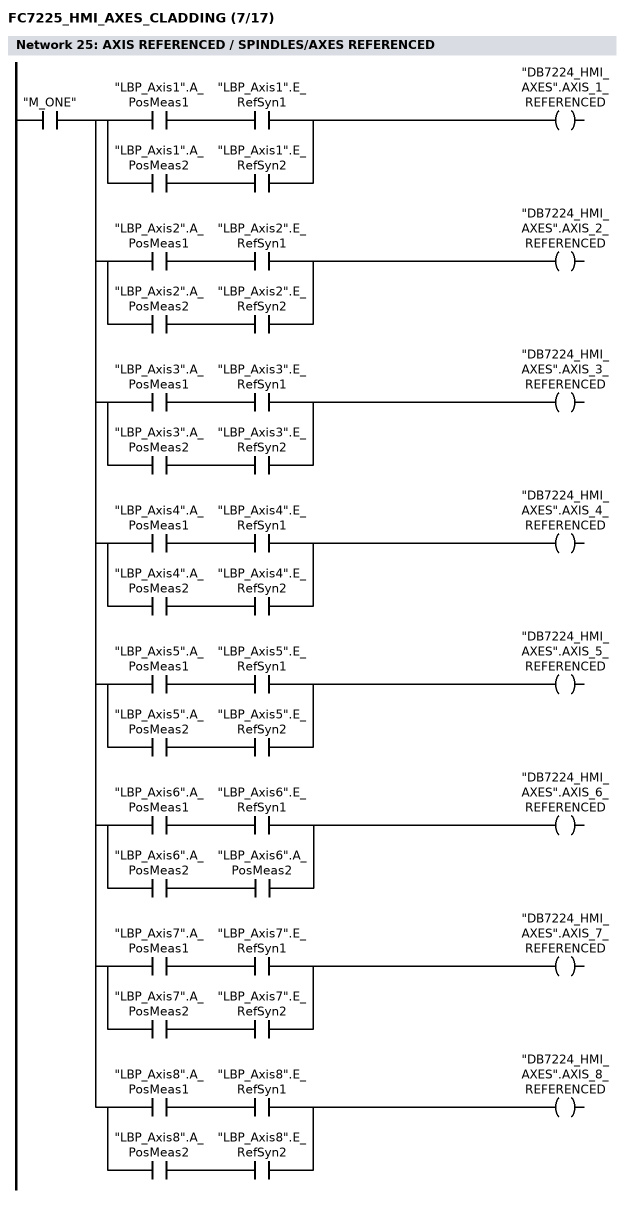
   RUNG wire#powerrail
      Contact( "M_ONE" )
      wire#w1
      Contact( "LBP_Axis1".A_PosMeas1 )
      Contact( "LBP_Axis1".E_RefSyn1 )
      wire#w2
      Coil( "DB7224_HMI_AXES".AXIS_1_REFERENCED )
   END_RUNG
   RUNG wire#w1
      Contact( "LBP_Axis1".A_PosMeas2 )
      Contact( "LBP_Axis1".E_RefSyn2 )
   END_RUNG wire#w2
   RUNG wire#w1
      Contact( "LBP_Axis2".A_PosMeas1 )
      Contact( "LBP_Axis2".E_RefSyn1 )
      wire#w3
      Coil( "DB7224_HMI_AXES".AXIS_2_REFERENCED )
   END_RUNG
   RUNG wire#w1
      Contact( "LBP_Axis2".A_PosMeas2 )
      Contact( "LBP_Axis2".E_RefSyn2 )
   END_RUNG wire#w3
   RUNG wire#w1
      Contact( "LBP_Axis3".A_PosMeas1 )
      Contact( "LBP_Axis3".E_RefSyn1 )
      wire#w4
      Coil( "DB7224_HMI_AXES".AXIS_3_REFERENCED )
   END_RUNG
   RUNG wire#w1
      Contact( "LBP_Axis3".A_PosMeas2 )
      Contact( "LBP_Axis3".E_RefSyn2 )
   END_RUNG wire#w4
   RUNG wire#w1
      Contact( "LBP_Axis4".A_PosMeas1 )
      Contact( "LBP_Axis4".E_RefSyn1 )
      wire#w5
      Coil( "DB7224_HMI_AXES".AXIS_4_REFERENCED )
   END_RUNG
   RUNG wire#w1
      Contact( "LBP_Axis4".A_PosMeas2 )
      Contact( "LBP_Axis4".E_RefSyn2 )
   END_RUNG wire#w5
   RUNG wire#w1
      Contact( "LBP_Axis5".A_PosMeas1 )
      Contact( "LBP_Axis5".E_RefSyn1 )
      wire#w6
      Coil( "DB7224_HMI_AXES".AXIS_5_REFERENCED )
   END_RUNG
   RUNG wire#w1
      Contact( "LBP_Axis5".A_PosMeas2 )
      Contact( "LBP_Axis5".E_RefSyn2 )
   END_RUNG wire#w6
   RUNG wire#w1
      Contact( "LBP_Axis6".A_PosMeas1 )
      Contact( "LBP_Axis6".E_RefSyn1 )
      wire#w7
      Coil( "DB7224_HMI_AXES".AXIS_6_REFERENCED )
   END_RUNG
   RUNG wire#w1
      Contact( "LBP_Axis6".A_PosMeas2 )
      Contact( "LBP_Axis6".A_PosMeas2 )
   END_RUNG wire#w7
   RUNG wire#w1
      Contact( "LBP_Axis7".A_PosMeas1 )
      Contact( "LBP_Axis7".E_RefSyn1 )
      wire#w8
      Coil( "DB7224_HMI_AXES".AXIS_7_REFERENCED )
   END_RUNG
   RUNG wire#w1
      Contact( "LBP_Axis7".A_PosMeas2 )
      Contact( "LBP_Axis7".E_RefSyn2 )
   END_RUNG wire#w8
   RUNG wire#w1
      Contact( "LBP_Axis8".A_PosMeas1 )
      Contact( "LBP_Axis8".E_RefSyn1 )
      wire#w9
      Coil( "DB7224_HMI_AXES".AXIS_8_REFERENCED )
   END_RUNG
   RUNG wire#w1
      Contact( "LBP_Axis8".A_PosMeas2 )
      Contact( "LBP_Axis8".E_RefSyn2 )
   END_RUNG wire#w9
   // the same network as SCL:
   "DB7224_HMI_AXES".AXIS_1_REFERENCED := "M_ONE" AND (("LBP_Axis1".A_PosMeas1 AND "LBP_Axis1".E_RefSyn1) OR ("LBP_Axis1".A_PosMeas2 AND "LBP_Axis1".E_RefSyn2));
   "DB7224_HMI_AXES".AXIS_2_REFERENCED := "M_ONE" AND (("LBP_Axis2".A_PosMeas1 AND "LBP_Axis2".E_RefSyn1) OR ("LBP_Axis2".A_PosMeas2 AND "LBP_Axis2".E_RefSyn2));
   "DB7224_HMI_AXES".AXIS_3_REFERENCED := "M_ONE" AND (("LBP_Axis3".A_PosMeas1 AND "LBP_Axis3".E_RefSyn1) OR ("LBP_Axis3".A_PosMeas2 AND "LBP_Axis3".E_RefSyn2));
   "DB7224_HMI_AXES".AXIS_4_REFERENCED := "M_ONE" AND (("LBP_Axis4".A_PosMeas1 AND "LBP_Axis4".E_RefSyn1) OR ("LBP_Axis4".A_PosMeas2 AND "LBP_Axis4".E_RefSyn2));
   "DB7224_HMI_AXES".AXIS_5_REFERENCED := "M_ONE" AND (("LBP_Axis5".A_PosMeas1 AND "LBP_Axis5".E_RefSyn1) OR ("LBP_Axis5".A_PosMeas2 AND "LBP_Axis5".E_RefSyn2));
   "DB7224_HMI_AXES".AXIS_6_REFERENCED := "M_ONE" AND (("LBP_Axis6".A_PosMeas1 AND "LBP_Axis6".E_RefSyn1) OR ("LBP_Axis6".A_PosMeas2 AND "LBP_Axis6".A_PosMeas2));
   "DB7224_HMI_AXES".AXIS_7_REFERENCED := "M_ONE" AND (("LBP_Axis7".A_PosMeas1 AND "LBP_Axis7".E_RefSyn1) OR ("LBP_Axis7".A_PosMeas2 AND "LBP_Axis7".E_RefSyn2));
   "DB7224_HMI_AXES".AXIS_8_REFERENCED := "M_ONE" AND (("LBP_Axis8".A_PosMeas1 AND "LBP_Axis8".E_RefSyn1) OR ("LBP_Axis8".A_PosMeas2 AND "LBP_Axis8".E_RefSyn2));
END_REGION

REGION Network 26: AXIS REFERENCED / AXES REFERENCED
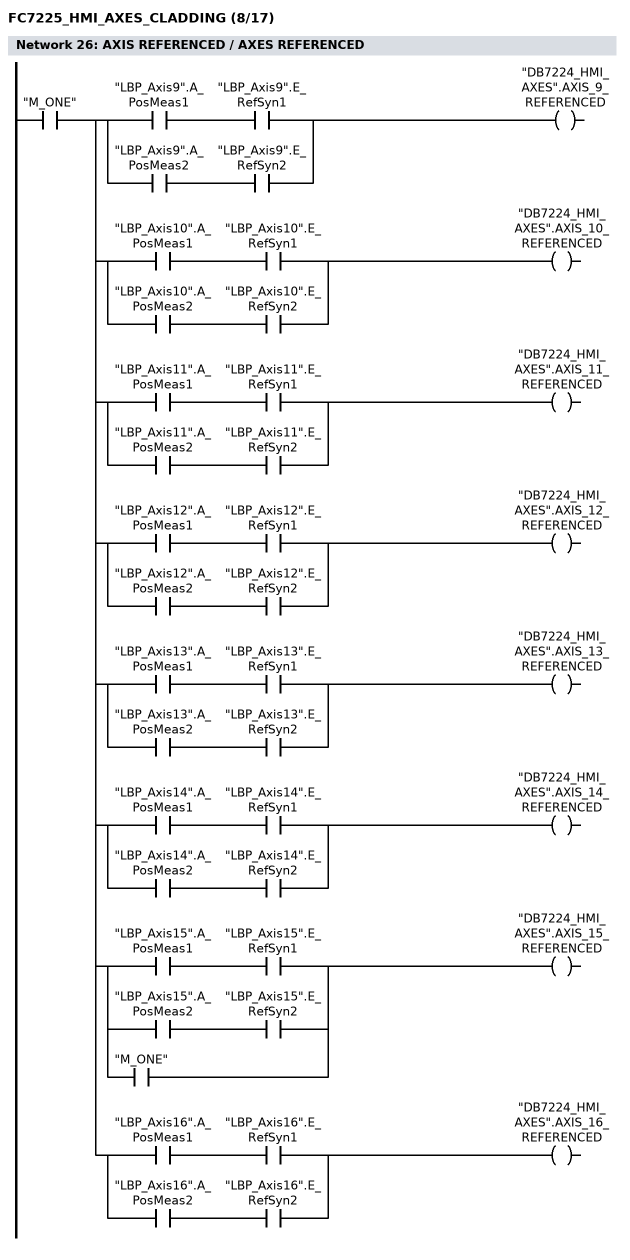
   RUNG wire#powerrail
      Contact( "M_ONE" )
      wire#w1
      Contact( "LBP_Axis9".A_PosMeas1 )
      Contact( "LBP_Axis9".E_RefSyn1 )
      wire#w2
      Coil( "DB7224_HMI_AXES".AXIS_9_REFERENCED )
   END_RUNG
   RUNG wire#w1
      Contact( "LBP_Axis9".A_PosMeas2 )
      Contact( "LBP_Axis9".E_RefSyn2 )
   END_RUNG wire#w2
   RUNG wire#w1
      Contact( "LBP_Axis10".A_PosMeas1 )
      Contact( "LBP_Axis10".E_RefSyn1 )
      wire#w3
      Coil( "DB7224_HMI_AXES".AXIS_10_REFERENCED )
   END_RUNG
   RUNG wire#w1
      Contact( "LBP_Axis10".A_PosMeas2 )
      Contact( "LBP_Axis10".E_RefSyn2 )
   END_RUNG wire#w3
   RUNG wire#w1
      Contact( "LBP_Axis11".A_PosMeas1 )
      Contact( "LBP_Axis11".E_RefSyn1 )
      wire#w4
      Coil( "DB7224_HMI_AXES".AXIS_11_REFERENCED )
   END_RUNG
   RUNG wire#w1
      Contact( "LBP_Axis11".A_PosMeas2 )
      Contact( "LBP_Axis11".E_RefSyn2 )
   END_RUNG wire#w4
   RUNG wire#w1
      Contact( "LBP_Axis12".A_PosMeas1 )
      Contact( "LBP_Axis12".E_RefSyn1 )
      wire#w5
      Coil( "DB7224_HMI_AXES".AXIS_12_REFERENCED )
   END_RUNG
   RUNG wire#w1
      Contact( "LBP_Axis12".A_PosMeas2 )
      Contact( "LBP_Axis12".E_RefSyn2 )
   END_RUNG wire#w5
   RUNG wire#w1
      Contact( "LBP_Axis13".A_PosMeas1 )
      Contact( "LBP_Axis13".E_RefSyn1 )
      wire#w6
      Coil( "DB7224_HMI_AXES".AXIS_13_REFERENCED )
   END_RUNG
   RUNG wire#w1
      Contact( "LBP_Axis13".A_PosMeas2 )
      Contact( "LBP_Axis13".E_RefSyn2 )
   END_RUNG wire#w6
   RUNG wire#w1
      Contact( "LBP_Axis14".A_PosMeas1 )
      Contact( "LBP_Axis14".E_RefSyn1 )
      wire#w7
      Coil( "DB7224_HMI_AXES".AXIS_14_REFERENCED )
   END_RUNG
   RUNG wire#w1
      Contact( "LBP_Axis14".A_PosMeas2 )
      Contact( "LBP_Axis14".E_RefSyn2 )
   END_RUNG wire#w7
   RUNG wire#w1
      Contact( "LBP_Axis15".A_PosMeas1 )
      Contact( "LBP_Axis15".E_RefSyn1 )
      wire#w8
      Coil( "DB7224_HMI_AXES".AXIS_15_REFERENCED )
   END_RUNG
   RUNG wire#w1
      Contact( "LBP_Axis15".A_PosMeas2 )
      Contact( "LBP_Axis15".E_RefSyn2 )
   END_RUNG wire#w8
   RUNG wire#w1
      Contact( "M_ONE" )
   END_RUNG wire#w8
   RUNG wire#w1
      Contact( "LBP_Axis16".A_PosMeas1 )
      Contact( "LBP_Axis16".E_RefSyn1 )
      wire#w9
      Coil( "DB7224_HMI_AXES".AXIS_16_REFERENCED )
   END_RUNG
   RUNG wire#w1
      Contact( "LBP_Axis16".A_PosMeas2 )
      Contact( "LBP_Axis16".E_RefSyn2 )
   END_RUNG wire#w9
   // the same network as SCL:
   "DB7224_HMI_AXES".AXIS_9_REFERENCED := "M_ONE" AND (("LBP_Axis9".A_PosMeas1 AND "LBP_Axis9".E_RefSyn1) OR ("LBP_Axis9".A_PosMeas2 AND "LBP_Axis9".E_RefSyn2));
   "DB7224_HMI_AXES".AXIS_10_REFERENCED := "M_ONE" AND (("LBP_Axis10".A_PosMeas1 AND "LBP_Axis10".E_RefSyn1) OR ("LBP_Axis10".A_PosMeas2 AND "LBP_Axis10".E_RefSyn2));
   "DB7224_HMI_AXES".AXIS_11_REFERENCED := "M_ONE" AND (("LBP_Axis11".A_PosMeas1 AND "LBP_Axis11".E_RefSyn1) OR ("LBP_Axis11".A_PosMeas2 AND "LBP_Axis11".E_RefSyn2));
   "DB7224_HMI_AXES".AXIS_12_REFERENCED := "M_ONE" AND (("LBP_Axis12".A_PosMeas1 AND "LBP_Axis12".E_RefSyn1) OR ("LBP_Axis12".A_PosMeas2 AND "LBP_Axis12".E_RefSyn2));
   "DB7224_HMI_AXES".AXIS_13_REFERENCED := "M_ONE" AND (("LBP_Axis13".A_PosMeas1 AND "LBP_Axis13".E_RefSyn1) OR ("LBP_Axis13".A_PosMeas2 AND "LBP_Axis13".E_RefSyn2));
   "DB7224_HMI_AXES".AXIS_14_REFERENCED := "M_ONE" AND (("LBP_Axis14".A_PosMeas1 AND "LBP_Axis14".E_RefSyn1) OR ("LBP_Axis14".A_PosMeas2 AND "LBP_Axis14".E_RefSyn2));
   "DB7224_HMI_AXES".AXIS_15_REFERENCED := "M_ONE" AND (("LBP_Axis15".A_PosMeas1 AND "LBP_Axis15".E_RefSyn1) OR ("LBP_Axis15".A_PosMeas2 AND "LBP_Axis15".E_RefSyn2) OR "M_ONE");
   "DB7224_HMI_AXES".AXIS_16_REFERENCED := "M_ONE" AND (("LBP_Axis16".A_PosMeas1 AND "LBP_Axis16".E_RefSyn1) OR ("LBP_Axis16".A_PosMeas2 AND "LBP_Axis16".E_RefSyn2));
END_REGION

REGION Network 27: AXIS REFERENCED / AXES REFERENCED
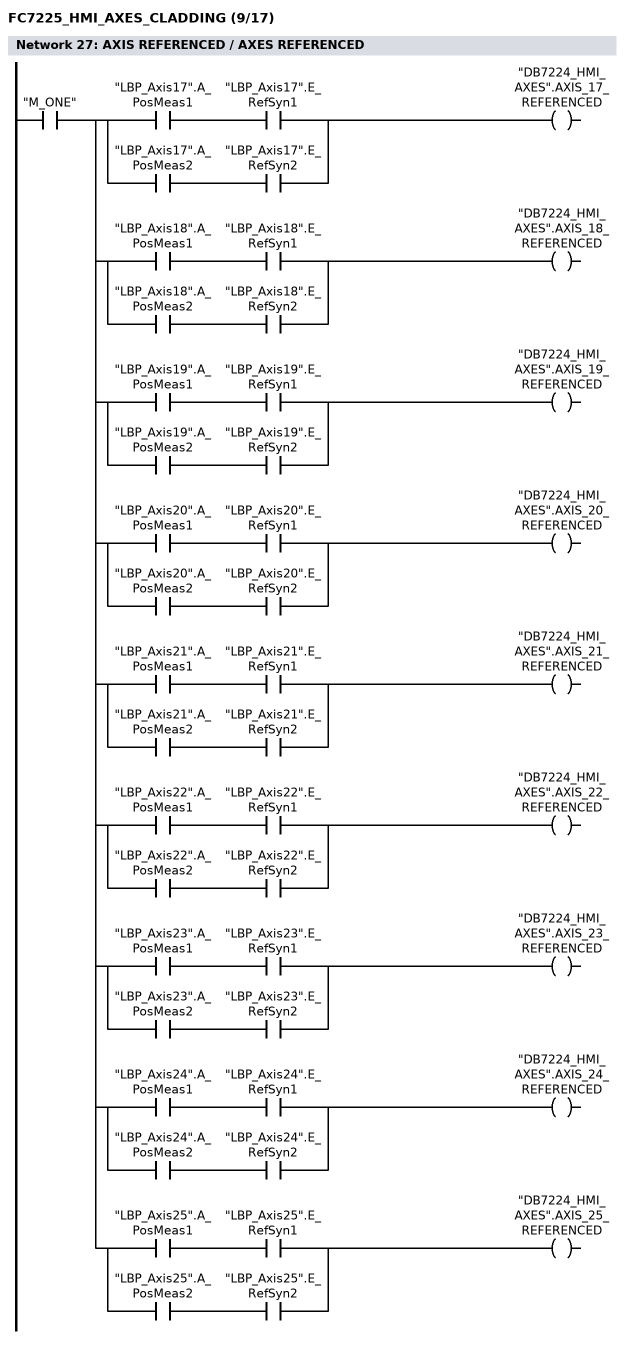
   RUNG wire#powerrail
      Contact( "M_ONE" )
      wire#w1
      Contact( "LBP_Axis17".A_PosMeas1 )
      Contact( "LBP_Axis17".E_RefSyn1 )
      wire#w2
      Coil( "DB7224_HMI_AXES".AXIS_17_REFERENCED )
   END_RUNG
   RUNG wire#w1
      Contact( "LBP_Axis17".A_PosMeas2 )
      Contact( "LBP_Axis17".E_RefSyn2 )
   END_RUNG wire#w2
   RUNG wire#w1
      Contact( "LBP_Axis18".A_PosMeas1 )
      Contact( "LBP_Axis18".E_RefSyn1 )
      wire#w3
      Coil( "DB7224_HMI_AXES".AXIS_18_REFERENCED )
   END_RUNG
   RUNG wire#w1
      Contact( "LBP_Axis18".A_PosMeas2 )
      Contact( "LBP_Axis18".E_RefSyn2 )
   END_RUNG wire#w3
   RUNG wire#w1
      Contact( "LBP_Axis19".A_PosMeas1 )
      Contact( "LBP_Axis19".E_RefSyn1 )
      wire#w4
      Coil( "DB7224_HMI_AXES".AXIS_19_REFERENCED )
   END_RUNG
   RUNG wire#w1
      Contact( "LBP_Axis19".A_PosMeas2 )
      Contact( "LBP_Axis19".E_RefSyn2 )
   END_RUNG wire#w4
   RUNG wire#w1
      Contact( "LBP_Axis20".A_PosMeas1 )
      Contact( "LBP_Axis20".E_RefSyn1 )
      wire#w5
      Coil( "DB7224_HMI_AXES".AXIS_20_REFERENCED )
   END_RUNG
   RUNG wire#w1
      Contact( "LBP_Axis20".A_PosMeas2 )
      Contact( "LBP_Axis20".E_RefSyn2 )
   END_RUNG wire#w5
   RUNG wire#w1
      Contact( "LBP_Axis21".A_PosMeas1 )
      Contact( "LBP_Axis21".E_RefSyn1 )
      wire#w6
      Coil( "DB7224_HMI_AXES".AXIS_21_REFERENCED )
   END_RUNG
   RUNG wire#w1
      Contact( "LBP_Axis21".A_PosMeas2 )
      Contact( "LBP_Axis21".E_RefSyn2 )
   END_RUNG wire#w6
   RUNG wire#w1
      Contact( "LBP_Axis22".A_PosMeas1 )
      Contact( "LBP_Axis22".E_RefSyn1 )
      wire#w7
      Coil( "DB7224_HMI_AXES".AXIS_22_REFERENCED )
   END_RUNG
   RUNG wire#w1
      Contact( "LBP_Axis22".A_PosMeas2 )
      Contact( "LBP_Axis22".E_RefSyn2 )
   END_RUNG wire#w7
   RUNG wire#w1
      Contact( "LBP_Axis23".A_PosMeas1 )
      Contact( "LBP_Axis23".E_RefSyn1 )
      wire#w8
      Coil( "DB7224_HMI_AXES".AXIS_23_REFERENCED )
   END_RUNG
   RUNG wire#w1
      Contact( "LBP_Axis23".A_PosMeas2 )
      Contact( "LBP_Axis23".E_RefSyn2 )
   END_RUNG wire#w8
   RUNG wire#w1
      Contact( "LBP_Axis24".A_PosMeas1 )
      Contact( "LBP_Axis24".E_RefSyn1 )
      wire#w9
      Coil( "DB7224_HMI_AXES".AXIS_24_REFERENCED )
   END_RUNG
   RUNG wire#w1
      Contact( "LBP_Axis24".A_PosMeas2 )
      Contact( "LBP_Axis24".E_RefSyn2 )
   END_RUNG wire#w9
   RUNG wire#w1
      Contact( "LBP_Axis25".A_PosMeas1 )
      Contact( "LBP_Axis25".E_RefSyn1 )
      wire#w10
      Coil( "DB7224_HMI_AXES".AXIS_25_REFERENCED )
   END_RUNG
   RUNG wire#w1
      Contact( "LBP_Axis25".A_PosMeas2 )
      Contact( "LBP_Axis25".E_RefSyn2 )
   END_RUNG wire#w10
   // the same network as SCL:
   "DB7224_HMI_AXES".AXIS_17_REFERENCED := "M_ONE" AND (("LBP_Axis17".A_PosMeas1 AND "LBP_Axis17".E_RefSyn1) OR ("LBP_Axis17".A_PosMeas2 AND "LBP_Axis17".E_RefSyn2));
   "DB7224_HMI_AXES".AXIS_18_REFERENCED := "M_ONE" AND (("LBP_Axis18".A_PosMeas1 AND "LBP_Axis18".E_RefSyn1) OR ("LBP_Axis18".A_PosMeas2 AND "LBP_Axis18".E_RefSyn2));
   "DB7224_HMI_AXES".AXIS_19_REFERENCED := "M_ONE" AND (("LBP_Axis19".A_PosMeas1 AND "LBP_Axis19".E_RefSyn1) OR ("LBP_Axis19".A_PosMeas2 AND "LBP_Axis19".E_RefSyn2));
   "DB7224_HMI_AXES".AXIS_20_REFERENCED := "M_ONE" AND (("LBP_Axis20".A_PosMeas1 AND "LBP_Axis20".E_RefSyn1) OR ("LBP_Axis20".A_PosMeas2 AND "LBP_Axis20".E_RefSyn2));
   "DB7224_HMI_AXES".AXIS_21_REFERENCED := "M_ONE" AND (("LBP_Axis21".A_PosMeas1 AND "LBP_Axis21".E_RefSyn1) OR ("LBP_Axis21".A_PosMeas2 AND "LBP_Axis21".E_RefSyn2));
   "DB7224_HMI_AXES".AXIS_22_REFERENCED := "M_ONE" AND (("LBP_Axis22".A_PosMeas1 AND "LBP_Axis22".E_RefSyn1) OR ("LBP_Axis22".A_PosMeas2 AND "LBP_Axis22".E_RefSyn2));
   "DB7224_HMI_AXES".AXIS_23_REFERENCED := "M_ONE" AND (("LBP_Axis23".A_PosMeas1 AND "LBP_Axis23".E_RefSyn1) OR ("LBP_Axis23".A_PosMeas2 AND "LBP_Axis23".E_RefSyn2));
   "DB7224_HMI_AXES".AXIS_24_REFERENCED := "M_ONE" AND (("LBP_Axis24".A_PosMeas1 AND "LBP_Axis24".E_RefSyn1) OR ("LBP_Axis24".A_PosMeas2 AND "LBP_Axis24".E_RefSyn2));
   "DB7224_HMI_AXES".AXIS_25_REFERENCED := "M_ONE" AND (("LBP_Axis25".A_PosMeas1 AND "LBP_Axis25".E_RefSyn1) OR ("LBP_Axis25".A_PosMeas2 AND "LBP_Axis25".E_RefSyn2));
END_REGION

REGION Network 28: AXIS REFERENCED / AXES REFERENCED
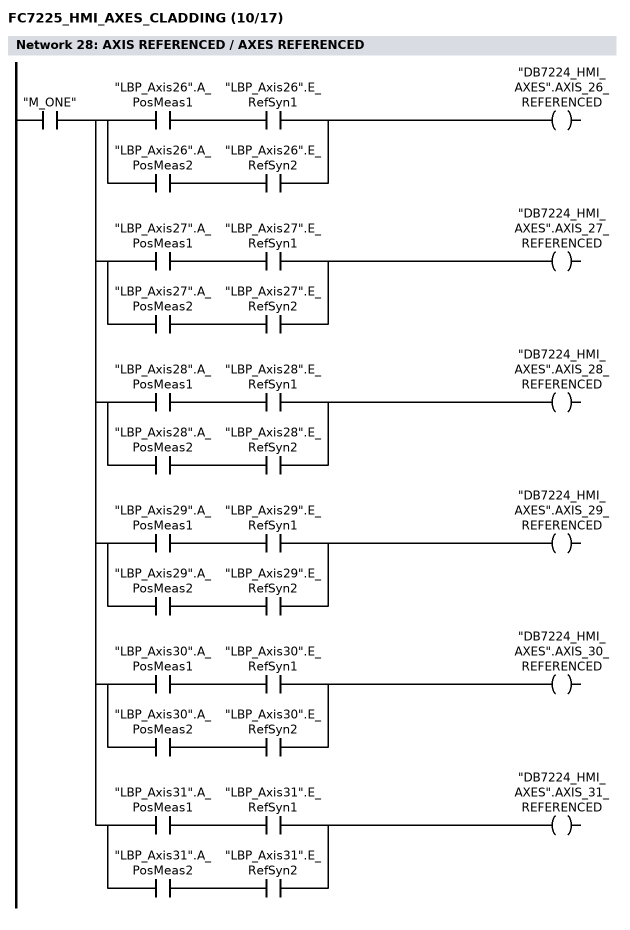
   RUNG wire#powerrail
      Contact( "M_ONE" )
      wire#w1
      Contact( "LBP_Axis26".A_PosMeas1 )
      Contact( "LBP_Axis26".E_RefSyn1 )
      wire#w2
      Coil( "DB7224_HMI_AXES".AXIS_26_REFERENCED )
   END_RUNG
   RUNG wire#w1
      Contact( "LBP_Axis26".A_PosMeas2 )
      Contact( "LBP_Axis26".E_RefSyn2 )
   END_RUNG wire#w2
   RUNG wire#w1
      Contact( "LBP_Axis27".A_PosMeas1 )
      Contact( "LBP_Axis27".E_RefSyn1 )
      wire#w3
      Coil( "DB7224_HMI_AXES".AXIS_27_REFERENCED )
   END_RUNG
   RUNG wire#w1
      Contact( "LBP_Axis27".A_PosMeas2 )
      Contact( "LBP_Axis27".E_RefSyn2 )
   END_RUNG wire#w3
   RUNG wire#w1
      Contact( "LBP_Axis28".A_PosMeas1 )
      Contact( "LBP_Axis28".E_RefSyn1 )
      wire#w4
      Coil( "DB7224_HMI_AXES".AXIS_28_REFERENCED )
   END_RUNG
   RUNG wire#w1
      Contact( "LBP_Axis28".A_PosMeas2 )
      Contact( "LBP_Axis28".E_RefSyn2 )
   END_RUNG wire#w4
   RUNG wire#w1
      Contact( "LBP_Axis29".A_PosMeas1 )
      Contact( "LBP_Axis29".E_RefSyn1 )
      wire#w5
      Coil( "DB7224_HMI_AXES".AXIS_29_REFERENCED )
   END_RUNG
   RUNG wire#w1
      Contact( "LBP_Axis29".A_PosMeas2 )
      Contact( "LBP_Axis29".E_RefSyn2 )
   END_RUNG wire#w5
   RUNG wire#w1
      Contact( "LBP_Axis30".A_PosMeas1 )
      Contact( "LBP_Axis30".E_RefSyn1 )
      wire#w6
      Coil( "DB7224_HMI_AXES".AXIS_30_REFERENCED )
   END_RUNG
   RUNG wire#w1
      Contact( "LBP_Axis30".A_PosMeas2 )
      Contact( "LBP_Axis30".E_RefSyn2 )
   END_RUNG wire#w6
   RUNG wire#w1
      Contact( "LBP_Axis31".A_PosMeas1 )
      Contact( "LBP_Axis31".E_RefSyn1 )
      wire#w7
      Coil( "DB7224_HMI_AXES".AXIS_31_REFERENCED )
   END_RUNG
   RUNG wire#w1
      Contact( "LBP_Axis31".A_PosMeas2 )
      Contact( "LBP_Axis31".E_RefSyn2 )
   END_RUNG wire#w7
   // the same network as SCL:
   "DB7224_HMI_AXES".AXIS_26_REFERENCED := "M_ONE" AND (("LBP_Axis26".A_PosMeas1 AND "LBP_Axis26".E_RefSyn1) OR ("LBP_Axis26".A_PosMeas2 AND "LBP_Axis26".E_RefSyn2));
   "DB7224_HMI_AXES".AXIS_27_REFERENCED := "M_ONE" AND (("LBP_Axis27".A_PosMeas1 AND "LBP_Axis27".E_RefSyn1) OR ("LBP_Axis27".A_PosMeas2 AND "LBP_Axis27".E_RefSyn2));
   "DB7224_HMI_AXES".AXIS_28_REFERENCED := "M_ONE" AND (("LBP_Axis28".A_PosMeas1 AND "LBP_Axis28".E_RefSyn1) OR ("LBP_Axis28".A_PosMeas2 AND "LBP_Axis28".E_RefSyn2));
   "DB7224_HMI_AXES".AXIS_29_REFERENCED := "M_ONE" AND (("LBP_Axis29".A_PosMeas1 AND "LBP_Axis29".E_RefSyn1) OR ("LBP_Axis29".A_PosMeas2 AND "LBP_Axis29".E_RefSyn2));
   "DB7224_HMI_AXES".AXIS_30_REFERENCED := "M_ONE" AND (("LBP_Axis30".A_PosMeas1 AND "LBP_Axis30".E_RefSyn1) OR ("LBP_Axis30".A_PosMeas2 AND "LBP_Axis30".E_RefSyn2));
   "DB7224_HMI_AXES".AXIS_31_REFERENCED := "M_ONE" AND (("LBP_Axis31".A_PosMeas1 AND "LBP_Axis31".E_RefSyn1) OR ("LBP_Axis31".A_PosMeas2 AND "LBP_Axis31".E_RefSyn2));
END_REGION

REGION Network 29: AXIS CONDITIONS / SPINDLE/AXES FEED HOLD CONDITIONS
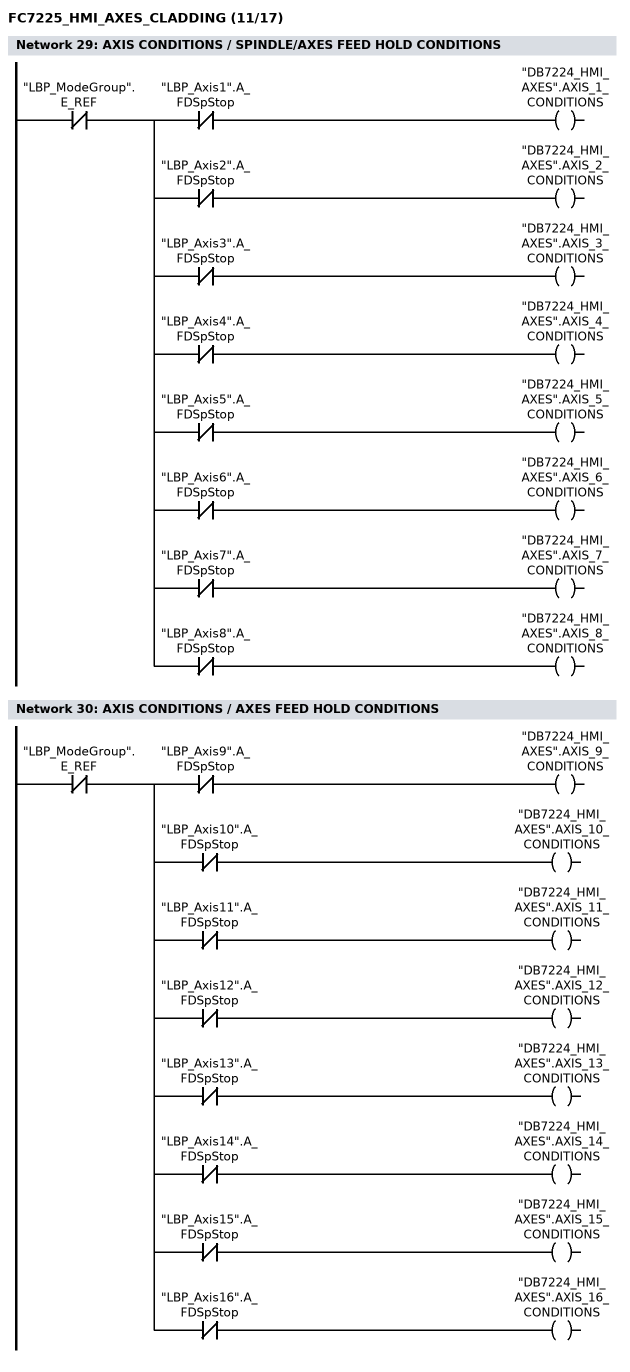
   RUNG wire#powerrail
      I_Contact( "LBP_ModeGroup".E_REF )
      wire#w1
      I_Contact( "LBP_Axis1".A_FDSpStop )
      Coil( "DB7224_HMI_AXES".AXIS_1_CONDITIONS )
   END_RUNG
   RUNG wire#w1
      I_Contact( "LBP_Axis2".A_FDSpStop )
      Coil( "DB7224_HMI_AXES".AXIS_2_CONDITIONS )
   END_RUNG
   RUNG wire#w1
      I_Contact( "LBP_Axis3".A_FDSpStop )
      Coil( "DB7224_HMI_AXES".AXIS_3_CONDITIONS )
   END_RUNG
   RUNG wire#w1
      I_Contact( "LBP_Axis4".A_FDSpStop )
      Coil( "DB7224_HMI_AXES".AXIS_4_CONDITIONS )
   END_RUNG
   RUNG wire#w1
      I_Contact( "LBP_Axis5".A_FDSpStop )
      Coil( "DB7224_HMI_AXES".AXIS_5_CONDITIONS )
   END_RUNG
   RUNG wire#w1
      I_Contact( "LBP_Axis6".A_FDSpStop )
      Coil( "DB7224_HMI_AXES".AXIS_6_CONDITIONS )
   END_RUNG
   RUNG wire#w1
      I_Contact( "LBP_Axis7".A_FDSpStop )
      Coil( "DB7224_HMI_AXES".AXIS_7_CONDITIONS )
   END_RUNG
   RUNG wire#w1
      I_Contact( "LBP_Axis8".A_FDSpStop )
      Coil( "DB7224_HMI_AXES".AXIS_8_CONDITIONS )
   END_RUNG
   // the same network as SCL:
   #_w1 := NOT "LBP_ModeGroup".E_REF;
   "DB7224_HMI_AXES".AXIS_1_CONDITIONS := #_w1 AND NOT "LBP_Axis1".A_FDSpStop;
   "DB7224_HMI_AXES".AXIS_2_CONDITIONS := #_w1 AND NOT "LBP_Axis2".A_FDSpStop;
   "DB7224_HMI_AXES".AXIS_3_CONDITIONS := #_w1 AND NOT "LBP_Axis3".A_FDSpStop;
   "DB7224_HMI_AXES".AXIS_4_CONDITIONS := #_w1 AND NOT "LBP_Axis4".A_FDSpStop;
   "DB7224_HMI_AXES".AXIS_5_CONDITIONS := #_w1 AND NOT "LBP_Axis5".A_FDSpStop;
   "DB7224_HMI_AXES".AXIS_6_CONDITIONS := #_w1 AND NOT "LBP_Axis6".A_FDSpStop;
   "DB7224_HMI_AXES".AXIS_7_CONDITIONS := #_w1 AND NOT "LBP_Axis7".A_FDSpStop;
   "DB7224_HMI_AXES".AXIS_8_CONDITIONS := #_w1 AND NOT "LBP_Axis8".A_FDSpStop;
END_REGION

REGION Network 30: AXIS CONDITIONS / AXES FEED HOLD CONDITIONS
   RUNG wire#powerrail
      I_Contact( "LBP_ModeGroup".E_REF )
      wire#w1
      I_Contact( "LBP_Axis9".A_FDSpStop )
      Coil( "DB7224_HMI_AXES".AXIS_9_CONDITIONS )
   END_RUNG
   RUNG wire#w1
      I_Contact( "LBP_Axis10".A_FDSpStop )
      Coil( "DB7224_HMI_AXES".AXIS_10_CONDITIONS )
   END_RUNG
   RUNG wire#w1
      I_Contact( "LBP_Axis11".A_FDSpStop )
      Coil( "DB7224_HMI_AXES".AXIS_11_CONDITIONS )
   END_RUNG
   RUNG wire#w1
      I_Contact( "LBP_Axis12".A_FDSpStop )
      Coil( "DB7224_HMI_AXES".AXIS_12_CONDITIONS )
   END_RUNG
   RUNG wire#w1
      I_Contact( "LBP_Axis13".A_FDSpStop )
      Coil( "DB7224_HMI_AXES".AXIS_13_CONDITIONS )
   END_RUNG
   RUNG wire#w1
      I_Contact( "LBP_Axis14".A_FDSpStop )
      Coil( "DB7224_HMI_AXES".AXIS_14_CONDITIONS )
   END_RUNG
   RUNG wire#w1
      I_Contact( "LBP_Axis15".A_FDSpStop )
      Coil( "DB7224_HMI_AXES".AXIS_15_CONDITIONS )
   END_RUNG
   RUNG wire#w1
      I_Contact( "LBP_Axis16".A_FDSpStop )
      Coil( "DB7224_HMI_AXES".AXIS_16_CONDITIONS )
   END_RUNG
   // the same network as SCL:
   #_w1 := NOT "LBP_ModeGroup".E_REF;
   "DB7224_HMI_AXES".AXIS_9_CONDITIONS := #_w1 AND NOT "LBP_Axis9".A_FDSpStop;
   "DB7224_HMI_AXES".AXIS_10_CONDITIONS := #_w1 AND NOT "LBP_Axis10".A_FDSpStop;
   "DB7224_HMI_AXES".AXIS_11_CONDITIONS := #_w1 AND NOT "LBP_Axis11".A_FDSpStop;
   "DB7224_HMI_AXES".AXIS_12_CONDITIONS := #_w1 AND NOT "LBP_Axis12".A_FDSpStop;
   "DB7224_HMI_AXES".AXIS_13_CONDITIONS := #_w1 AND NOT "LBP_Axis13".A_FDSpStop;
   "DB7224_HMI_AXES".AXIS_14_CONDITIONS := #_w1 AND NOT "LBP_Axis14".A_FDSpStop;
   "DB7224_HMI_AXES".AXIS_15_CONDITIONS := #_w1 AND NOT "LBP_Axis15".A_FDSpStop;
   "DB7224_HMI_AXES".AXIS_16_CONDITIONS := #_w1 AND NOT "LBP_Axis16".A_FDSpStop;
END_REGION

REGION Network 31: AXIS CONDITIONS / AXES FEED HOLD CONDITIONS
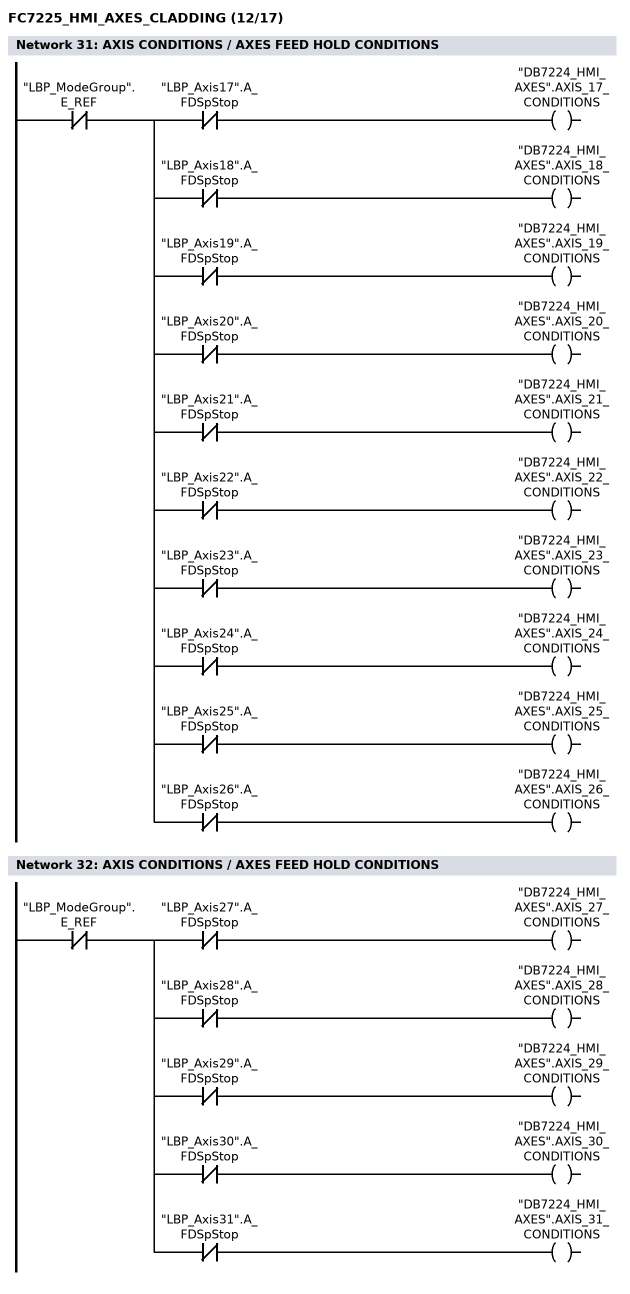
   RUNG wire#powerrail
      I_Contact( "LBP_ModeGroup".E_REF )
      wire#w1
      I_Contact( "LBP_Axis17".A_FDSpStop )
      Coil( "DB7224_HMI_AXES".AXIS_17_CONDITIONS )
   END_RUNG
   RUNG wire#w1
      I_Contact( "LBP_Axis18".A_FDSpStop )
      Coil( "DB7224_HMI_AXES".AXIS_18_CONDITIONS )
   END_RUNG
   RUNG wire#w1
      I_Contact( "LBP_Axis19".A_FDSpStop )
      Coil( "DB7224_HMI_AXES".AXIS_19_CONDITIONS )
   END_RUNG
   RUNG wire#w1
      I_Contact( "LBP_Axis20".A_FDSpStop )
      Coil( "DB7224_HMI_AXES".AXIS_20_CONDITIONS )
   END_RUNG
   RUNG wire#w1
      I_Contact( "LBP_Axis21".A_FDSpStop )
      Coil( "DB7224_HMI_AXES".AXIS_21_CONDITIONS )
   END_RUNG
   RUNG wire#w1
      I_Contact( "LBP_Axis22".A_FDSpStop )
      Coil( "DB7224_HMI_AXES".AXIS_22_CONDITIONS )
   END_RUNG
   RUNG wire#w1
      I_Contact( "LBP_Axis23".A_FDSpStop )
      Coil( "DB7224_HMI_AXES".AXIS_23_CONDITIONS )
   END_RUNG
   RUNG wire#w1
      I_Contact( "LBP_Axis24".A_FDSpStop )
      Coil( "DB7224_HMI_AXES".AXIS_24_CONDITIONS )
   END_RUNG
   RUNG wire#w1
      I_Contact( "LBP_Axis25".A_FDSpStop )
      Coil( "DB7224_HMI_AXES".AXIS_25_CONDITIONS )
   END_RUNG
   RUNG wire#w1
      I_Contact( "LBP_Axis26".A_FDSpStop )
      Coil( "DB7224_HMI_AXES".AXIS_26_CONDITIONS )
   END_RUNG
   // the same network as SCL:
   #_w1 := NOT "LBP_ModeGroup".E_REF;
   "DB7224_HMI_AXES".AXIS_17_CONDITIONS := #_w1 AND NOT "LBP_Axis17".A_FDSpStop;
   "DB7224_HMI_AXES".AXIS_18_CONDITIONS := #_w1 AND NOT "LBP_Axis18".A_FDSpStop;
   "DB7224_HMI_AXES".AXIS_19_CONDITIONS := #_w1 AND NOT "LBP_Axis19".A_FDSpStop;
   "DB7224_HMI_AXES".AXIS_20_CONDITIONS := #_w1 AND NOT "LBP_Axis20".A_FDSpStop;
   "DB7224_HMI_AXES".AXIS_21_CONDITIONS := #_w1 AND NOT "LBP_Axis21".A_FDSpStop;
   "DB7224_HMI_AXES".AXIS_22_CONDITIONS := #_w1 AND NOT "LBP_Axis22".A_FDSpStop;
   "DB7224_HMI_AXES".AXIS_23_CONDITIONS := #_w1 AND NOT "LBP_Axis23".A_FDSpStop;
   "DB7224_HMI_AXES".AXIS_24_CONDITIONS := #_w1 AND NOT "LBP_Axis24".A_FDSpStop;
   "DB7224_HMI_AXES".AXIS_25_CONDITIONS := #_w1 AND NOT "LBP_Axis25".A_FDSpStop;
   "DB7224_HMI_AXES".AXIS_26_CONDITIONS := #_w1 AND NOT "LBP_Axis26".A_FDSpStop;
END_REGION

REGION Network 32: AXIS CONDITIONS / AXES FEED HOLD CONDITIONS
   RUNG wire#powerrail
      I_Contact( "LBP_ModeGroup".E_REF )
      wire#w1
      I_Contact( "LBP_Axis27".A_FDSpStop )
      Coil( "DB7224_HMI_AXES".AXIS_27_CONDITIONS )
   END_RUNG
   RUNG wire#w1
      I_Contact( "LBP_Axis28".A_FDSpStop )
      Coil( "DB7224_HMI_AXES".AXIS_28_CONDITIONS )
   END_RUNG
   RUNG wire#w1
      I_Contact( "LBP_Axis29".A_FDSpStop )
      Coil( "DB7224_HMI_AXES".AXIS_29_CONDITIONS )
   END_RUNG
   RUNG wire#w1
      I_Contact( "LBP_Axis30".A_FDSpStop )
      Coil( "DB7224_HMI_AXES".AXIS_30_CONDITIONS )
   END_RUNG
   RUNG wire#w1
      I_Contact( "LBP_Axis31".A_FDSpStop )
      Coil( "DB7224_HMI_AXES".AXIS_31_CONDITIONS )
   END_RUNG
   // the same network as SCL:
   #_w1 := NOT "LBP_ModeGroup".E_REF;
   "DB7224_HMI_AXES".AXIS_27_CONDITIONS := #_w1 AND NOT "LBP_Axis27".A_FDSpStop;
   "DB7224_HMI_AXES".AXIS_28_CONDITIONS := #_w1 AND NOT "LBP_Axis28".A_FDSpStop;
   "DB7224_HMI_AXES".AXIS_29_CONDITIONS := #_w1 AND NOT "LBP_Axis29".A_FDSpStop;
   "DB7224_HMI_AXES".AXIS_30_CONDITIONS := #_w1 AND NOT "LBP_Axis30".A_FDSpStop;
   "DB7224_HMI_AXES".AXIS_31_CONDITIONS := #_w1 AND NOT "LBP_Axis31".A_FDSpStop;
END_REGION

REGION Network 33: BA3 LIST SELECTED CHANNEL / BA3 SELECTED UNITS
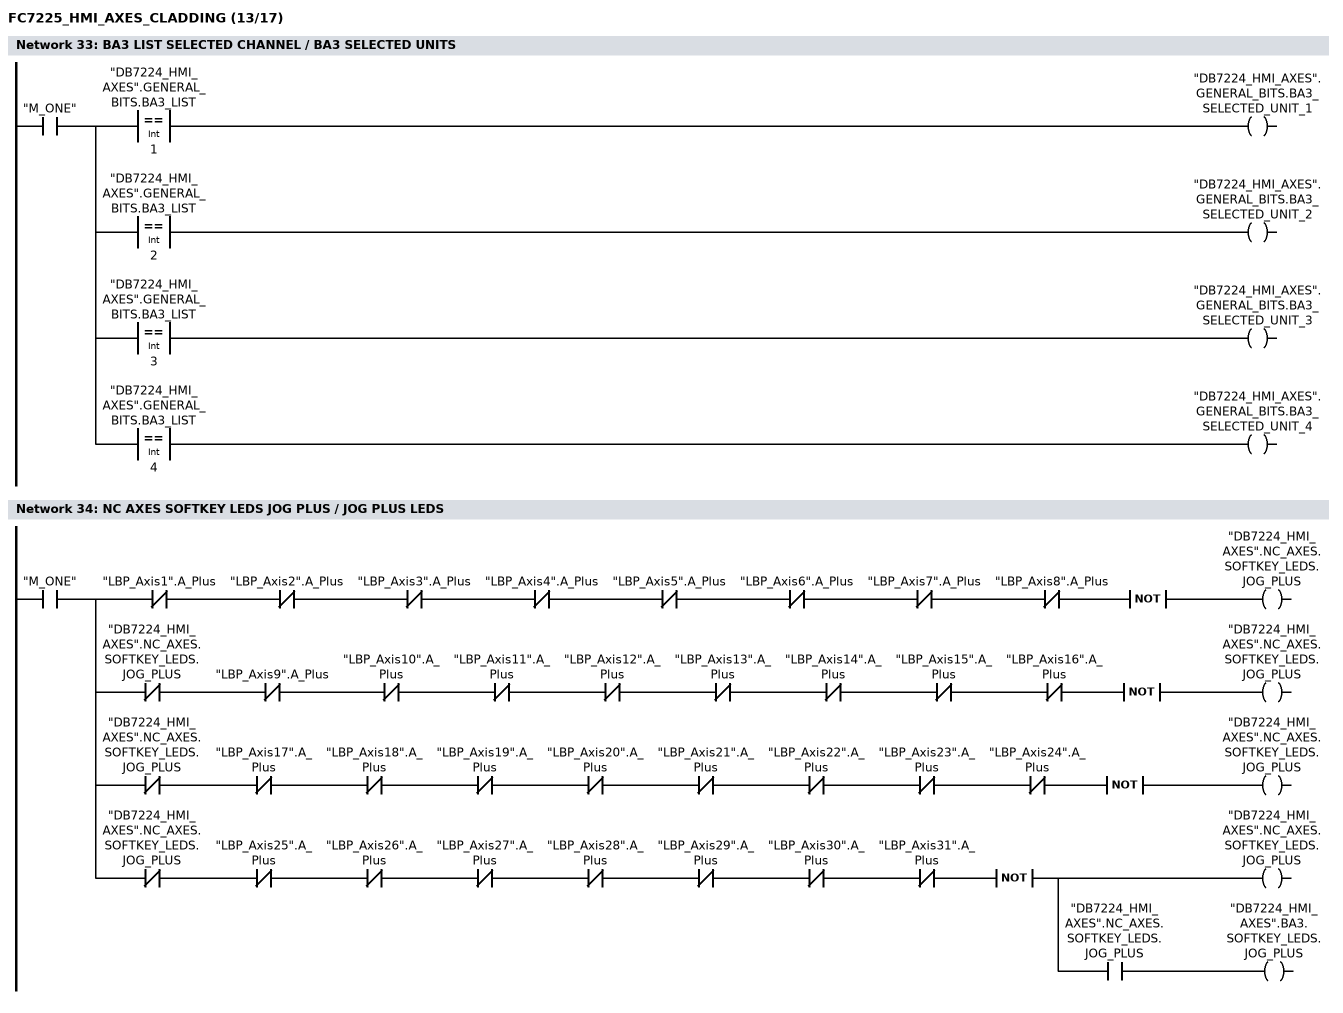
   RUNG wire#powerrail
      Contact( "M_ONE" )
      wire#w1
      { S7_Templates := "SrcType := Int" } EQ_Contact(in1 := "DB7224_HMI_AXES".GENERAL_BITS.BA3_LIST, in2 := 1)
      Coil( "DB7224_HMI_AXES".GENERAL_BITS.BA3_SELECTED_UNIT_1 )
   END_RUNG
   RUNG wire#w1
      { S7_Templates := "SrcType := Int" } EQ_Contact(in1 := "DB7224_HMI_AXES".GENERAL_BITS.BA3_LIST, in2 := 2)
      Coil( "DB7224_HMI_AXES".GENERAL_BITS.BA3_SELECTED_UNIT_2 )
   END_RUNG
   RUNG wire#w1
      { S7_Templates := "SrcType := Int" } EQ_Contact(in1 := "DB7224_HMI_AXES".GENERAL_BITS.BA3_LIST, in2 := 3)
      Coil( "DB7224_HMI_AXES".GENERAL_BITS.BA3_SELECTED_UNIT_3 )
   END_RUNG
   RUNG wire#w1
      { S7_Templates := "SrcType := Int" } EQ_Contact(in1 := "DB7224_HMI_AXES".GENERAL_BITS.BA3_LIST, in2 := 4)
      Coil( "DB7224_HMI_AXES".GENERAL_BITS.BA3_SELECTED_UNIT_4 )
   END_RUNG
   // the same network as SCL:
   "DB7224_HMI_AXES".GENERAL_BITS.BA3_SELECTED_UNIT_1 := "M_ONE" AND ("DB7224_HMI_AXES".GENERAL_BITS.BA3_LIST = 1);
   "DB7224_HMI_AXES".GENERAL_BITS.BA3_SELECTED_UNIT_2 := "M_ONE" AND ("DB7224_HMI_AXES".GENERAL_BITS.BA3_LIST = 2);
   "DB7224_HMI_AXES".GENERAL_BITS.BA3_SELECTED_UNIT_3 := "M_ONE" AND ("DB7224_HMI_AXES".GENERAL_BITS.BA3_LIST = 3);
   "DB7224_HMI_AXES".GENERAL_BITS.BA3_SELECTED_UNIT_4 := "M_ONE" AND ("DB7224_HMI_AXES".GENERAL_BITS.BA3_LIST = 4);
END_REGION

REGION Network 34: NC AXES SOFTKEY LEDS JOG PLUS / JOG PLUS LEDS
   RUNG wire#powerrail
      Contact( "M_ONE" )
      wire#w1
      I_Contact( "LBP_Axis1".A_Plus )
      I_Contact( "LBP_Axis2".A_Plus )
      I_Contact( "LBP_Axis3".A_Plus )
      I_Contact( "LBP_Axis4".A_Plus )
      I_Contact( "LBP_Axis5".A_Plus )
      I_Contact( "LBP_Axis6".A_Plus )
      I_Contact( "LBP_Axis7".A_Plus )
      I_Contact( "LBP_Axis8".A_Plus )
      Not()
      Coil( "DB7224_HMI_AXES".NC_AXES.SOFTKEY_LEDS.JOG_PLUS )
   END_RUNG
   RUNG wire#w1
      I_Contact( "DB7224_HMI_AXES".NC_AXES.SOFTKEY_LEDS.JOG_PLUS )
      I_Contact( "LBP_Axis9".A_Plus )
      I_Contact( "LBP_Axis10".A_Plus )
      I_Contact( "LBP_Axis11".A_Plus )
      I_Contact( "LBP_Axis12".A_Plus )
      I_Contact( "LBP_Axis13".A_Plus )
      I_Contact( "LBP_Axis14".A_Plus )
      I_Contact( "LBP_Axis15".A_Plus )
      I_Contact( "LBP_Axis16".A_Plus )
      Not()
      Coil( "DB7224_HMI_AXES".NC_AXES.SOFTKEY_LEDS.JOG_PLUS )
   END_RUNG
   RUNG wire#w1
      I_Contact( "DB7224_HMI_AXES".NC_AXES.SOFTKEY_LEDS.JOG_PLUS )
      I_Contact( "LBP_Axis17".A_Plus )
      I_Contact( "LBP_Axis18".A_Plus )
      I_Contact( "LBP_Axis19".A_Plus )
      I_Contact( "LBP_Axis20".A_Plus )
      I_Contact( "LBP_Axis21".A_Plus )
      I_Contact( "LBP_Axis22".A_Plus )
      I_Contact( "LBP_Axis23".A_Plus )
      I_Contact( "LBP_Axis24".A_Plus )
      Not()
      Coil( "DB7224_HMI_AXES".NC_AXES.SOFTKEY_LEDS.JOG_PLUS )
   END_RUNG
   RUNG wire#w1
      I_Contact( "DB7224_HMI_AXES".NC_AXES.SOFTKEY_LEDS.JOG_PLUS )
      I_Contact( "LBP_Axis25".A_Plus )
      I_Contact( "LBP_Axis26".A_Plus )
      I_Contact( "LBP_Axis27".A_Plus )
      I_Contact( "LBP_Axis28".A_Plus )
      I_Contact( "LBP_Axis29".A_Plus )
      I_Contact( "LBP_Axis30".A_Plus )
      I_Contact( "LBP_Axis31".A_Plus )
      Not()
      wire#w2
      Coil( "DB7224_HMI_AXES".NC_AXES.SOFTKEY_LEDS.JOG_PLUS )
   END_RUNG
   RUNG wire#w2
      Contact( "DB7224_HMI_AXES".NC_AXES.SOFTKEY_LEDS.JOG_PLUS )
      Coil( "DB7224_HMI_AXES".BA3.SOFTKEY_LEDS.JOG_PLUS )
   END_RUNG
   // the same network as SCL:
   "DB7224_HMI_AXES".NC_AXES.SOFTKEY_LEDS.JOG_PLUS := NOT ("M_ONE" AND NOT "LBP_Axis1".A_Plus AND NOT "LBP_Axis2".A_Plus AND NOT "LBP_Axis3".A_Plus AND NOT "LBP_Axis4".A_Plus AND NOT "LBP_Axis5".A_Plus AND NOT "LBP_Axis6".A_Plus AND NOT "LBP_Axis7".A_Plus AND NOT "LBP_Axis8".A_Plus);
   "DB7224_HMI_AXES".NC_AXES.SOFTKEY_LEDS.JOG_PLUS := NOT ("M_ONE" AND NOT "DB7224_HMI_AXES".NC_AXES.SOFTKEY_LEDS.JOG_PLUS AND NOT "LBP_Axis9".A_Plus AND NOT "LBP_Axis10".A_Plus AND NOT "LBP_Axis11".A_Plus AND NOT "LBP_Axis12".A_Plus AND NOT "LBP_Axis13".A_Plus AND NOT "LBP_Axis14".A_Plus AND NOT "LBP_Axis15".A_Plus AND NOT "LBP_Axis16".A_Plus);
   "DB7224_HMI_AXES".NC_AXES.SOFTKEY_LEDS.JOG_PLUS := NOT ("M_ONE" AND NOT "DB7224_HMI_AXES".NC_AXES.SOFTKEY_LEDS.JOG_PLUS AND NOT "LBP_Axis17".A_Plus AND NOT "LBP_Axis18".A_Plus AND NOT "LBP_Axis19".A_Plus AND NOT "LBP_Axis20".A_Plus AND NOT "LBP_Axis21".A_Plus AND NOT "LBP_Axis22".A_Plus AND NOT "LBP_Axis23".A_Plus AND NOT "LBP_Axis24".A_Plus);
   "DB7224_HMI_AXES".NC_AXES.SOFTKEY_LEDS.JOG_PLUS := NOT ("M_ONE" AND NOT "DB7224_HMI_AXES".NC_AXES.SOFTKEY_LEDS.JOG_PLUS AND NOT "LBP_Axis25".A_Plus AND NOT "LBP_Axis26".A_Plus AND NOT "LBP_Axis27".A_Plus AND NOT "LBP_Axis28".A_Plus AND NOT "LBP_Axis29".A_Plus AND NOT "LBP_Axis30".A_Plus AND NOT "LBP_Axis31".A_Plus);
   "DB7224_HMI_AXES".BA3.SOFTKEY_LEDS.JOG_PLUS := "DB7224_HMI_AXES".NC_AXES.SOFTKEY_LEDS.JOG_PLUS AND "DB7224_HMI_AXES".NC_AXES.SOFTKEY_LEDS.JOG_PLUS;
END_REGION

REGION Network 35: NC AXES SOFTKEY LEDS JOG MINUS / JOG MINUS LEDS
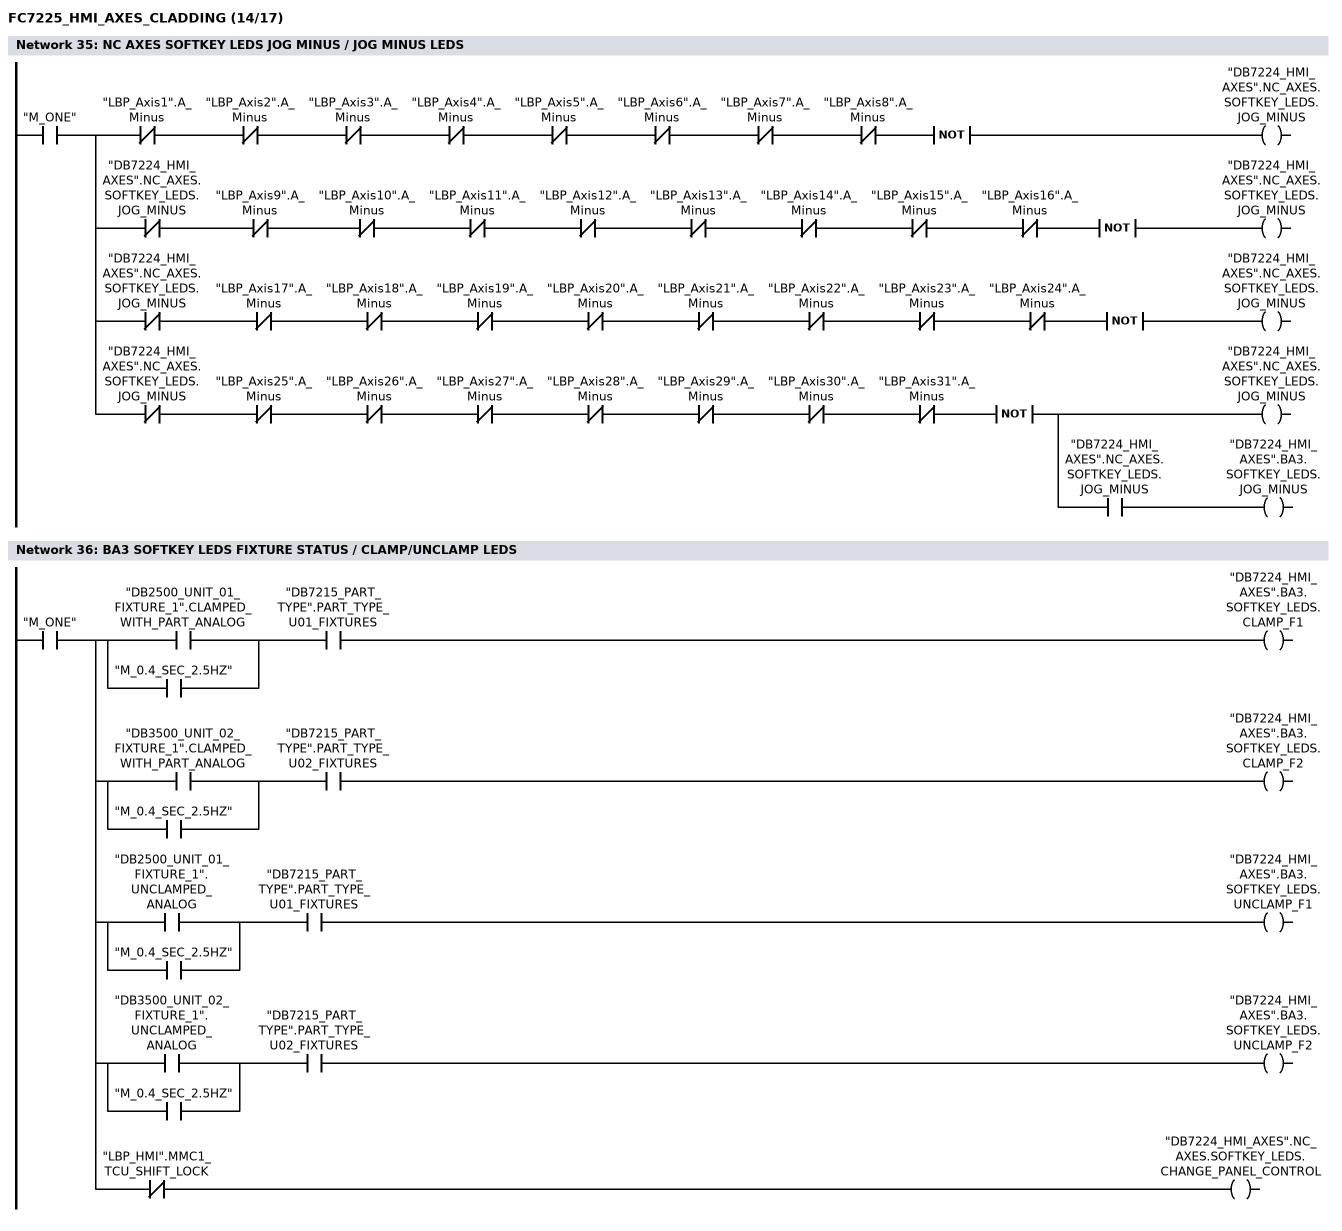
   RUNG wire#powerrail
      Contact( "M_ONE" )
      wire#w1
      I_Contact( "LBP_Axis1".A_Minus )
      I_Contact( "LBP_Axis2".A_Minus )
      I_Contact( "LBP_Axis3".A_Minus )
      I_Contact( "LBP_Axis4".A_Minus )
      I_Contact( "LBP_Axis5".A_Minus )
      I_Contact( "LBP_Axis6".A_Minus )
      I_Contact( "LBP_Axis7".A_Minus )
      I_Contact( "LBP_Axis8".A_Minus )
      Not()
      Coil( "DB7224_HMI_AXES".NC_AXES.SOFTKEY_LEDS.JOG_MINUS )
   END_RUNG
   RUNG wire#w1
      I_Contact( "DB7224_HMI_AXES".NC_AXES.SOFTKEY_LEDS.JOG_MINUS )
      I_Contact( "LBP_Axis9".A_Minus )
      I_Contact( "LBP_Axis10".A_Minus )
      I_Contact( "LBP_Axis11".A_Minus )
      I_Contact( "LBP_Axis12".A_Minus )
      I_Contact( "LBP_Axis13".A_Minus )
      I_Contact( "LBP_Axis14".A_Minus )
      I_Contact( "LBP_Axis15".A_Minus )
      I_Contact( "LBP_Axis16".A_Minus )
      Not()
      Coil( "DB7224_HMI_AXES".NC_AXES.SOFTKEY_LEDS.JOG_MINUS )
   END_RUNG
   RUNG wire#w1
      I_Contact( "DB7224_HMI_AXES".NC_AXES.SOFTKEY_LEDS.JOG_MINUS )
      I_Contact( "LBP_Axis17".A_Minus )
      I_Contact( "LBP_Axis18".A_Minus )
      I_Contact( "LBP_Axis19".A_Minus )
      I_Contact( "LBP_Axis20".A_Minus )
      I_Contact( "LBP_Axis21".A_Minus )
      I_Contact( "LBP_Axis22".A_Minus )
      I_Contact( "LBP_Axis23".A_Minus )
      I_Contact( "LBP_Axis24".A_Minus )
      Not()
      Coil( "DB7224_HMI_AXES".NC_AXES.SOFTKEY_LEDS.JOG_MINUS )
   END_RUNG
   RUNG wire#w1
      I_Contact( "DB7224_HMI_AXES".NC_AXES.SOFTKEY_LEDS.JOG_MINUS )
      I_Contact( "LBP_Axis25".A_Minus )
      I_Contact( "LBP_Axis26".A_Minus )
      I_Contact( "LBP_Axis27".A_Minus )
      I_Contact( "LBP_Axis28".A_Minus )
      I_Contact( "LBP_Axis29".A_Minus )
      I_Contact( "LBP_Axis30".A_Minus )
      I_Contact( "LBP_Axis31".A_Minus )
      Not()
      wire#w2
      Coil( "DB7224_HMI_AXES".NC_AXES.SOFTKEY_LEDS.JOG_MINUS )
   END_RUNG
   RUNG wire#w2
      Contact( "DB7224_HMI_AXES".NC_AXES.SOFTKEY_LEDS.JOG_MINUS )
      Coil( "DB7224_HMI_AXES".BA3.SOFTKEY_LEDS.JOG_MINUS )
   END_RUNG
   // the same network as SCL:
   "DB7224_HMI_AXES".NC_AXES.SOFTKEY_LEDS.JOG_MINUS := NOT ("M_ONE" AND NOT "LBP_Axis1".A_Minus AND NOT "LBP_Axis2".A_Minus AND NOT "LBP_Axis3".A_Minus AND NOT "LBP_Axis4".A_Minus AND NOT "LBP_Axis5".A_Minus AND NOT "LBP_Axis6".A_Minus AND NOT "LBP_Axis7".A_Minus AND NOT "LBP_Axis8".A_Minus);
   "DB7224_HMI_AXES".NC_AXES.SOFTKEY_LEDS.JOG_MINUS := NOT ("M_ONE" AND NOT "DB7224_HMI_AXES".NC_AXES.SOFTKEY_LEDS.JOG_MINUS AND NOT "LBP_Axis9".A_Minus AND NOT "LBP_Axis10".A_Minus AND NOT "LBP_Axis11".A_Minus AND NOT "LBP_Axis12".A_Minus AND NOT "LBP_Axis13".A_Minus AND NOT "LBP_Axis14".A_Minus AND NOT "LBP_Axis15".A_Minus AND NOT "LBP_Axis16".A_Minus);
   "DB7224_HMI_AXES".NC_AXES.SOFTKEY_LEDS.JOG_MINUS := NOT ("M_ONE" AND NOT "DB7224_HMI_AXES".NC_AXES.SOFTKEY_LEDS.JOG_MINUS AND NOT "LBP_Axis17".A_Minus AND NOT "LBP_Axis18".A_Minus AND NOT "LBP_Axis19".A_Minus AND NOT "LBP_Axis20".A_Minus AND NOT "LBP_Axis21".A_Minus AND NOT "LBP_Axis22".A_Minus AND NOT "LBP_Axis23".A_Minus AND NOT "LBP_Axis24".A_Minus);
   "DB7224_HMI_AXES".NC_AXES.SOFTKEY_LEDS.JOG_MINUS := NOT ("M_ONE" AND NOT "DB7224_HMI_AXES".NC_AXES.SOFTKEY_LEDS.JOG_MINUS AND NOT "LBP_Axis25".A_Minus AND NOT "LBP_Axis26".A_Minus AND NOT "LBP_Axis27".A_Minus AND NOT "LBP_Axis28".A_Minus AND NOT "LBP_Axis29".A_Minus AND NOT "LBP_Axis30".A_Minus AND NOT "LBP_Axis31".A_Minus);
   "DB7224_HMI_AXES".BA3.SOFTKEY_LEDS.JOG_MINUS := "DB7224_HMI_AXES".NC_AXES.SOFTKEY_LEDS.JOG_MINUS AND "DB7224_HMI_AXES".NC_AXES.SOFTKEY_LEDS.JOG_MINUS;
END_REGION

REGION Network 36: BA3 SOFTKEY LEDS FIXTURE STATUS / CLAMP/UNCLAMP LEDS
   RUNG wire#powerrail
      Contact( "M_ONE" )
      wire#w1
      Contact( "DB2500_UNIT_01_FIXTURE_1".CLAMPED_WITH_PART_ANALOG )
      wire#w2
      Contact( "DB7215_PART_TYPE".PART_TYPE_U01_FIXTURES )
      Coil( "DB7224_HMI_AXES".BA3.SOFTKEY_LEDS.CLAMP_F1 )
   END_RUNG
   RUNG wire#w1
      Contact( "M_0.4_SEC_2.5HZ" )
   END_RUNG wire#w2
   RUNG wire#w1
      Contact( "DB3500_UNIT_02_FIXTURE_1".CLAMPED_WITH_PART_ANALOG )
      wire#w3
      Contact( "DB7215_PART_TYPE".PART_TYPE_U02_FIXTURES )
      Coil( "DB7224_HMI_AXES".BA3.SOFTKEY_LEDS.CLAMP_F2 )
   END_RUNG
   RUNG wire#w1
      Contact( "M_0.4_SEC_2.5HZ" )
   END_RUNG wire#w3
   RUNG wire#w1
      Contact( "DB2500_UNIT_01_FIXTURE_1".UNCLAMPED_ANALOG )
      wire#w4
      Contact( "DB7215_PART_TYPE".PART_TYPE_U01_FIXTURES )
      Coil( "DB7224_HMI_AXES".BA3.SOFTKEY_LEDS.UNCLAMP_F1 )
   END_RUNG
   RUNG wire#w1
      Contact( "M_0.4_SEC_2.5HZ" )
   END_RUNG wire#w4
   RUNG wire#w1
      Contact( "DB3500_UNIT_02_FIXTURE_1".UNCLAMPED_ANALOG )
      wire#w5
      Contact( "DB7215_PART_TYPE".PART_TYPE_U02_FIXTURES )
      Coil( "DB7224_HMI_AXES".BA3.SOFTKEY_LEDS.UNCLAMP_F2 )
   END_RUNG
   RUNG wire#w1
      Contact( "M_0.4_SEC_2.5HZ" )
   END_RUNG wire#w5
   RUNG wire#w1
      I_Contact( "LBP_HMI".MMC1_TCU_SHIFT_LOCK )
      Coil( "DB7224_HMI_AXES".NC_AXES.SOFTKEY_LEDS.CHANGE_PANEL_CONTROL )
   END_RUNG
   // the same network as SCL:
   "DB7224_HMI_AXES".BA3.SOFTKEY_LEDS.CLAMP_F1 := "M_ONE" AND ("DB2500_UNIT_01_FIXTURE_1".CLAMPED_WITH_PART_ANALOG OR "M_0.4_SEC_2.5HZ") AND "DB7215_PART_TYPE".PART_TYPE_U01_FIXTURES;
   "DB7224_HMI_AXES".BA3.SOFTKEY_LEDS.CLAMP_F2 := "M_ONE" AND ("DB3500_UNIT_02_FIXTURE_1".CLAMPED_WITH_PART_ANALOG OR "M_0.4_SEC_2.5HZ") AND "DB7215_PART_TYPE".PART_TYPE_U02_FIXTURES;
   "DB7224_HMI_AXES".BA3.SOFTKEY_LEDS.UNCLAMP_F1 := "M_ONE" AND ("DB2500_UNIT_01_FIXTURE_1".UNCLAMPED_ANALOG OR "M_0.4_SEC_2.5HZ") AND "DB7215_PART_TYPE".PART_TYPE_U01_FIXTURES;
   "DB7224_HMI_AXES".BA3.SOFTKEY_LEDS.UNCLAMP_F2 := "M_ONE" AND ("DB3500_UNIT_02_FIXTURE_1".UNCLAMPED_ANALOG OR "M_0.4_SEC_2.5HZ") AND "DB7215_PART_TYPE".PART_TYPE_U02_FIXTURES;
   "DB7224_HMI_AXES".NC_AXES.SOFTKEY_LEDS.CHANGE_PANEL_CONTROL := "M_ONE" AND NOT "LBP_HMI".MMC1_TCU_SHIFT_LOCK;
END_REGION

REGION Network 37: NC AXES SOFTKEY LEDS SPINDLES SBH SG / SPINDLES SBH/SG LED
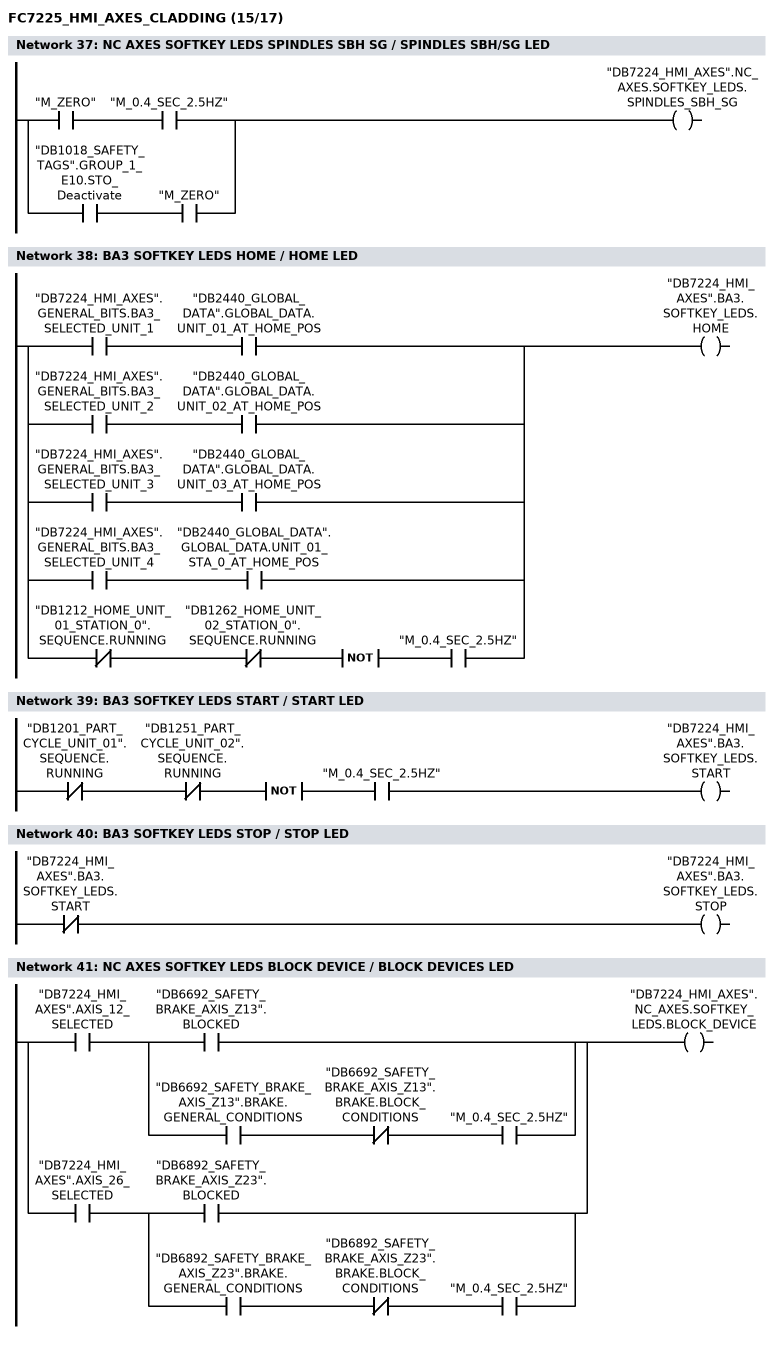
   RUNG wire#powerrail
      Contact( "M_ZERO" )
      Contact( "M_0.4_SEC_2.5HZ" )
      wire#w1
      Coil( "DB7224_HMI_AXES".NC_AXES.SOFTKEY_LEDS.SPINDLES_SBH_SG )
   END_RUNG
   RUNG wire#powerrail
      Contact( "DB1018_SAFETY_TAGS".GROUP_1_E10.STO_Deactivate )
      Contact( "M_ZERO" )
   END_RUNG wire#w1
   // the same network as SCL:
   "DB7224_HMI_AXES".NC_AXES.SOFTKEY_LEDS.SPINDLES_SBH_SG := ("M_ZERO" AND "M_0.4_SEC_2.5HZ") OR ("DB1018_SAFETY_TAGS".GROUP_1_E10.STO_Deactivate AND "M_ZERO");
END_REGION

REGION Network 38: BA3 SOFTKEY LEDS HOME / HOME LED
   RUNG wire#powerrail
      Contact( "DB7224_HMI_AXES".GENERAL_BITS.BA3_SELECTED_UNIT_1 )
      Contact( "DB2440_GLOBAL_DATA".GLOBAL_DATA.UNIT_01_AT_HOME_POS )
      wire#w1
      Coil( "DB7224_HMI_AXES".BA3.SOFTKEY_LEDS.HOME )
   END_RUNG
   RUNG wire#powerrail
      Contact( "DB7224_HMI_AXES".GENERAL_BITS.BA3_SELECTED_UNIT_2 )
      Contact( "DB2440_GLOBAL_DATA".GLOBAL_DATA.UNIT_02_AT_HOME_POS )
   END_RUNG wire#w1
   RUNG wire#powerrail
      Contact( "DB7224_HMI_AXES".GENERAL_BITS.BA3_SELECTED_UNIT_3 )
      Contact( "DB2440_GLOBAL_DATA".GLOBAL_DATA.UNIT_03_AT_HOME_POS )
   END_RUNG wire#w1
   RUNG wire#powerrail
      Contact( "DB7224_HMI_AXES".GENERAL_BITS.BA3_SELECTED_UNIT_4 )
      Contact( "DB2440_GLOBAL_DATA".GLOBAL_DATA.UNIT_01_STA_0_AT_HOME_POS )
   END_RUNG wire#w1
   RUNG wire#powerrail
      I_Contact( "DB1212_HOME_UNIT_01_STATION_0".SEQUENCE.RUNNING )
      I_Contact( "DB1262_HOME_UNIT_02_STATION_0".SEQUENCE.RUNNING )
      Not()
      Contact( "M_0.4_SEC_2.5HZ" )
   END_RUNG wire#w1
   // the same network as SCL:
   "DB7224_HMI_AXES".BA3.SOFTKEY_LEDS.HOME := ("DB7224_HMI_AXES".GENERAL_BITS.BA3_SELECTED_UNIT_1 AND "DB2440_GLOBAL_DATA".GLOBAL_DATA.UNIT_01_AT_HOME_POS) OR ("DB7224_HMI_AXES".GENERAL_BITS.BA3_SELECTED_UNIT_2 AND "DB2440_GLOBAL_DATA".GLOBAL_DATA.UNIT_02_AT_HOME_POS) OR ("DB7224_HMI_AXES".GENERAL_BITS.BA3_SELECTED_UNIT_3 AND "DB2440_GLOBAL_DATA".GLOBAL_DATA.UNIT_03_AT_HOME_POS) OR ("DB7224_HMI_AXES".GENERAL_BITS.BA3_SELECTED_UNIT_4 AND "DB2440_GLOBAL_DATA".GLOBAL_DATA.UNIT_01_STA_0_AT_HOME_POS) OR (NOT (NOT "DB1212_HOME_UNIT_01_STATION_0".SEQUENCE.RUNNING AND NOT "DB1262_HOME_UNIT_02_STATION_0".SEQUENCE.RUNNING) AND "M_0.4_SEC_2.5HZ");
END_REGION

REGION Network 39: BA3 SOFTKEY LEDS START / START LED
   RUNG wire#powerrail
      I_Contact( "DB1201_PART_CYCLE_UNIT_01".SEQUENCE.RUNNING )
      I_Contact( "DB1251_PART_CYCLE_UNIT_02".SEQUENCE.RUNNING )
      Not()
      Contact( "M_0.4_SEC_2.5HZ" )
      Coil( "DB7224_HMI_AXES".BA3.SOFTKEY_LEDS.START )
   END_RUNG
   // the same network as SCL:
   "DB7224_HMI_AXES".BA3.SOFTKEY_LEDS.START := NOT (NOT "DB1201_PART_CYCLE_UNIT_01".SEQUENCE.RUNNING AND NOT "DB1251_PART_CYCLE_UNIT_02".SEQUENCE.RUNNING) AND "M_0.4_SEC_2.5HZ";
END_REGION

REGION Network 40: BA3 SOFTKEY LEDS STOP / STOP LED
   RUNG wire#powerrail
      I_Contact( "DB7224_HMI_AXES".BA3.SOFTKEY_LEDS.START )
      Coil( "DB7224_HMI_AXES".BA3.SOFTKEY_LEDS.STOP )
   END_RUNG
   // the same network as SCL:
   "DB7224_HMI_AXES".BA3.SOFTKEY_LEDS.STOP := NOT "DB7224_HMI_AXES".BA3.SOFTKEY_LEDS.START;
END_REGION

REGION Network 41: NC AXES SOFTKEY LEDS BLOCK DEVICE / BLOCK DEVICES LED
   RUNG wire#powerrail
      Contact( "DB7224_HMI_AXES".AXIS_12_SELECTED )
      wire#w1
      Contact( "DB6692_SAFETY_BRAKE_AXIS_Z13".BLOCKED )
      wire#w2
      Coil( "DB7224_HMI_AXES".NC_AXES.SOFTKEY_LEDS.BLOCK_DEVICE )
   END_RUNG
   RUNG wire#w1
      Contact( "DB6692_SAFETY_BRAKE_AXIS_Z13".BRAKE.GENERAL_CONDITIONS )
      I_Contact( "DB6692_SAFETY_BRAKE_AXIS_Z13".BRAKE.BLOCK_CONDITIONS )
      Contact( "M_0.4_SEC_2.5HZ" )
   END_RUNG wire#w2
   RUNG wire#powerrail
      Contact( "DB7224_HMI_AXES".AXIS_26_SELECTED )
      wire#w3
      Contact( "DB6892_SAFETY_BRAKE_AXIS_Z23".BLOCKED )
   END_RUNG wire#w2
   RUNG wire#w3
      Contact( "DB6892_SAFETY_BRAKE_AXIS_Z23".BRAKE.GENERAL_CONDITIONS )
      I_Contact( "DB6892_SAFETY_BRAKE_AXIS_Z23".BRAKE.BLOCK_CONDITIONS )
      Contact( "M_0.4_SEC_2.5HZ" )
   END_RUNG wire#w2
   // the same network as SCL:
   "DB7224_HMI_AXES".NC_AXES.SOFTKEY_LEDS.BLOCK_DEVICE := ("DB7224_HMI_AXES".AXIS_12_SELECTED AND ("DB6692_SAFETY_BRAKE_AXIS_Z13".BLOCKED OR ("DB6692_SAFETY_BRAKE_AXIS_Z13".BRAKE.GENERAL_CONDITIONS AND NOT "DB6692_SAFETY_BRAKE_AXIS_Z13".BRAKE.BLOCK_CONDITIONS AND "M_0.4_SEC_2.5HZ"))) OR ("DB7224_HMI_AXES".AXIS_26_SELECTED AND ("DB6892_SAFETY_BRAKE_AXIS_Z23".BLOCKED OR ("DB6892_SAFETY_BRAKE_AXIS_Z23".BRAKE.GENERAL_CONDITIONS AND NOT "DB6892_SAFETY_BRAKE_AXIS_Z23".BRAKE.BLOCK_CONDITIONS AND "M_0.4_SEC_2.5HZ")));
END_REGION

REGION Network 42: NC AXES SOFTKEY LEDS UNBLOCK DEVICE / UNBLOCK DEVICES LED
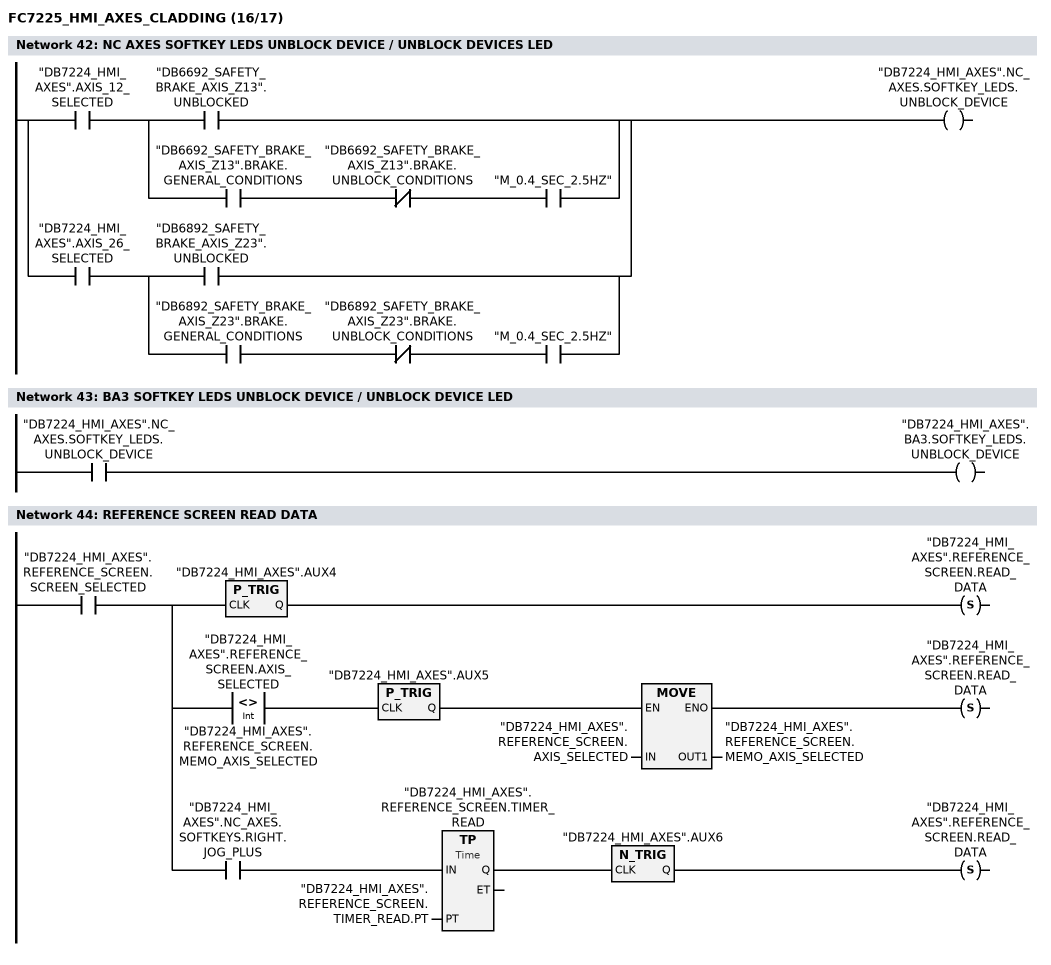
   RUNG wire#powerrail
      Contact( "DB7224_HMI_AXES".AXIS_12_SELECTED )
      wire#w1
      Contact( "DB6692_SAFETY_BRAKE_AXIS_Z13".UNBLOCKED )
      wire#w2
      Coil( "DB7224_HMI_AXES".NC_AXES.SOFTKEY_LEDS.UNBLOCK_DEVICE )
   END_RUNG
   RUNG wire#w1
      Contact( "DB6692_SAFETY_BRAKE_AXIS_Z13".BRAKE.GENERAL_CONDITIONS )
      I_Contact( "DB6692_SAFETY_BRAKE_AXIS_Z13".BRAKE.UNBLOCK_CONDITIONS )
      Contact( "M_0.4_SEC_2.5HZ" )
   END_RUNG wire#w2
   RUNG wire#powerrail
      Contact( "DB7224_HMI_AXES".AXIS_26_SELECTED )
      wire#w3
      Contact( "DB6892_SAFETY_BRAKE_AXIS_Z23".UNBLOCKED )
   END_RUNG wire#w2
   RUNG wire#w3
      Contact( "DB6892_SAFETY_BRAKE_AXIS_Z23".BRAKE.GENERAL_CONDITIONS )
      I_Contact( "DB6892_SAFETY_BRAKE_AXIS_Z23".BRAKE.UNBLOCK_CONDITIONS )
      Contact( "M_0.4_SEC_2.5HZ" )
   END_RUNG wire#w2
   // the same network as SCL:
   "DB7224_HMI_AXES".NC_AXES.SOFTKEY_LEDS.UNBLOCK_DEVICE := ("DB7224_HMI_AXES".AXIS_12_SELECTED AND ("DB6692_SAFETY_BRAKE_AXIS_Z13".UNBLOCKED OR ("DB6692_SAFETY_BRAKE_AXIS_Z13".BRAKE.GENERAL_CONDITIONS AND NOT "DB6692_SAFETY_BRAKE_AXIS_Z13".BRAKE.UNBLOCK_CONDITIONS AND "M_0.4_SEC_2.5HZ"))) OR ("DB7224_HMI_AXES".AXIS_26_SELECTED AND ("DB6892_SAFETY_BRAKE_AXIS_Z23".UNBLOCKED OR ("DB6892_SAFETY_BRAKE_AXIS_Z23".BRAKE.GENERAL_CONDITIONS AND NOT "DB6892_SAFETY_BRAKE_AXIS_Z23".BRAKE.UNBLOCK_CONDITIONS AND "M_0.4_SEC_2.5HZ")));
END_REGION

REGION Network 43: BA3 SOFTKEY LEDS UNBLOCK DEVICE / UNBLOCK DEVICE LED
   RUNG wire#powerrail
      Contact( "DB7224_HMI_AXES".NC_AXES.SOFTKEY_LEDS.UNBLOCK_DEVICE )
      Coil( "DB7224_HMI_AXES".BA3.SOFTKEY_LEDS.UNBLOCK_DEVICE )
   END_RUNG
   // the same network as SCL:
   "DB7224_HMI_AXES".BA3.SOFTKEY_LEDS.UNBLOCK_DEVICE := "DB7224_HMI_AXES".NC_AXES.SOFTKEY_LEDS.UNBLOCK_DEVICE;
END_REGION

REGION Network 44: REFERENCE SCREEN READ DATA
   RUNG wire#powerrail
      Contact( "DB7224_HMI_AXES".REFERENCE_SCREEN.SCREEN_SELECTED )
      wire#w1
      P_Trig( "DB7224_HMI_AXES".AUX4 )
      S_Coil( "DB7224_HMI_AXES".REFERENCE_SCREEN.READ_DATA )
   END_RUNG
   RUNG wire#w1
      { S7_Templates := "SrcType := Int" } NE_Contact(in1 := "DB7224_HMI_AXES".REFERENCE_SCREEN.AXIS_SELECTED, in2 := "DB7224_HMI_AXES".REFERENCE_SCREEN.MEMO_AXIS_SELECTED)
      P_Trig( "DB7224_HMI_AXES".AUX5 )
      Move(in := "DB7224_HMI_AXES".REFERENCE_SCREEN.AXIS_SELECTED, out1 => "DB7224_HMI_AXES".REFERENCE_SCREEN.MEMO_AXIS_SELECTED)
      S_Coil( "DB7224_HMI_AXES".REFERENCE_SCREEN.READ_DATA )
   END_RUNG
   RUNG wire#w1
      Contact( "DB7224_HMI_AXES".NC_AXES.SOFTKEYS.RIGHT.JOG_PLUS )
      { S7_Templates := "time_type := Time" } "DB7224_HMI_AXES".REFERENCE_SCREEN.TIMER_READ.TP(pt := "DB7224_HMI_AXES".REFERENCE_SCREEN.TIMER_READ.PT, et =>)
      N_Trig( "DB7224_HMI_AXES".AUX6 )
      S_Coil( "DB7224_HMI_AXES".REFERENCE_SCREEN.READ_DATA )
   END_RUNG
   // the same network as SCL:
   #_w1 := "DB7224_HMI_AXES".REFERENCE_SCREEN.SCREEN_SELECTED AND NOT "DB7224_HMI_AXES".AUX4;   // rising edge
   "DB7224_HMI_AXES".AUX4 := "DB7224_HMI_AXES".REFERENCE_SCREEN.SCREEN_SELECTED;
   IF #_w1 THEN "DB7224_HMI_AXES".REFERENCE_SCREEN.READ_DATA := TRUE; END_IF;
   #_w2 := "DB7224_HMI_AXES".REFERENCE_SCREEN.SCREEN_SELECTED AND ("DB7224_HMI_AXES".REFERENCE_SCREEN.AXIS_SELECTED <> "DB7224_HMI_AXES".REFERENCE_SCREEN.MEMO_AXIS_SELECTED);
   #_w3 := #_w2 AND NOT "DB7224_HMI_AXES".AUX5;   // rising edge
   "DB7224_HMI_AXES".AUX5 := #_w2;
   IF #_w3 THEN
       "DB7224_HMI_AXES".REFERENCE_SCREEN.MEMO_AXIS_SELECTED := "DB7224_HMI_AXES".REFERENCE_SCREEN.AXIS_SELECTED;
       "DB7224_HMI_AXES".REFERENCE_SCREEN.READ_DATA := TRUE;
   END_IF;
   "DB7224_HMI_AXES".REFERENCE_SCREEN.TIMER_READ.TP(IN := "DB7224_HMI_AXES".REFERENCE_SCREEN.SCREEN_SELECTED AND "DB7224_HMI_AXES".NC_AXES.SOFTKEYS.RIGHT.JOG_PLUS,
                           PT := "DB7224_HMI_AXES".REFERENCE_SCREEN.TIMER_READ.PT);
   #_w4 := NOT "DB7224_HMI_AXES".REFERENCE_SCREEN.TIMER_READ.Q AND "DB7224_HMI_AXES".AUX6;   // falling edge
   "DB7224_HMI_AXES".AUX6 := "DB7224_HMI_AXES".REFERENCE_SCREEN.TIMER_READ.Q;
   IF #_w4 THEN "DB7224_HMI_AXES".REFERENCE_SCREEN.READ_DATA := TRUE; END_IF;
END_REGION

REGION Network 45: AXIS OVERRIDE MG2
   // OVERRIDE VALUE 26=100%, 9=75%, 15=50%, 7=25%, 1=0%
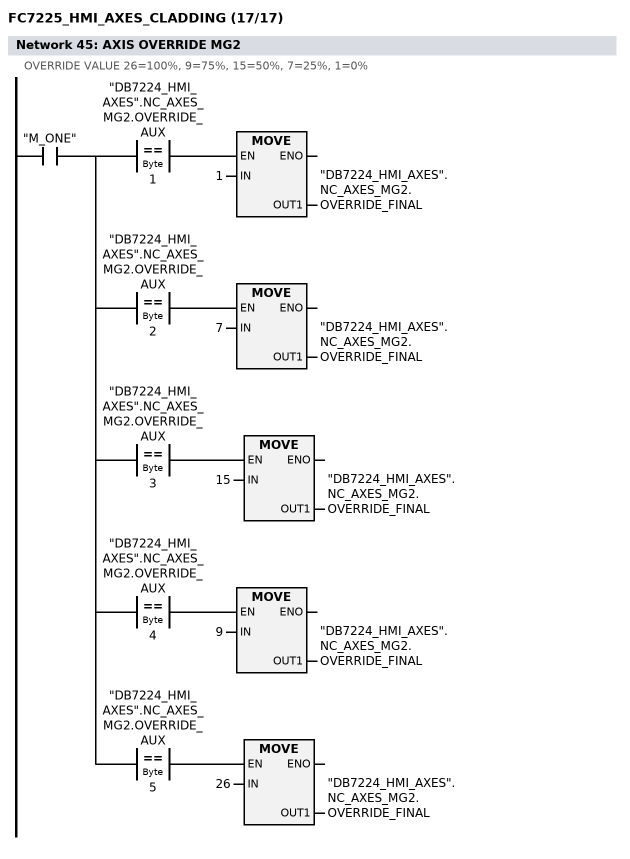
   RUNG wire#powerrail
      Contact( "M_ONE" )
      wire#w1
      { S7_Templates := "SrcType := Byte" } EQ_Contact(in1 := "DB7224_HMI_AXES".NC_AXES_MG2.OVERRIDE_AUX, in2 := 1)
      Move(in := 1, out1 => "DB7224_HMI_AXES".NC_AXES_MG2.OVERRIDE_FINAL)
   END_RUNG
   RUNG wire#w1
      { S7_Templates := "SrcType := Byte" } EQ_Contact(in1 := "DB7224_HMI_AXES".NC_AXES_MG2.OVERRIDE_AUX, in2 := 2)
      Move(in := 7, out1 => "DB7224_HMI_AXES".NC_AXES_MG2.OVERRIDE_FINAL)
   END_RUNG
   RUNG wire#w1
      { S7_Templates := "SrcType := Byte" } EQ_Contact(in1 := "DB7224_HMI_AXES".NC_AXES_MG2.OVERRIDE_AUX, in2 := 3)
      Move(in := 15, out1 => "DB7224_HMI_AXES".NC_AXES_MG2.OVERRIDE_FINAL)
   END_RUNG
   RUNG wire#w1
      { S7_Templates := "SrcType := Byte" } EQ_Contact(in1 := "DB7224_HMI_AXES".NC_AXES_MG2.OVERRIDE_AUX, in2 := 4)
      Move(in := 9, out1 => "DB7224_HMI_AXES".NC_AXES_MG2.OVERRIDE_FINAL)
   END_RUNG
   RUNG wire#w1
      { S7_Templates := "SrcType := Byte" } EQ_Contact(in1 := "DB7224_HMI_AXES".NC_AXES_MG2.OVERRIDE_AUX, in2 := 5)
      Move(in := 26, out1 => "DB7224_HMI_AXES".NC_AXES_MG2.OVERRIDE_FINAL)
   END_RUNG
   // the same network as SCL:
   IF "M_ONE" AND ("DB7224_HMI_AXES".NC_AXES_MG2.OVERRIDE_AUX = 1) THEN
       "DB7224_HMI_AXES".NC_AXES_MG2.OVERRIDE_FINAL := 1;
   END_IF;
   IF "M_ONE" AND ("DB7224_HMI_AXES".NC_AXES_MG2.OVERRIDE_AUX = 2) THEN
       "DB7224_HMI_AXES".NC_AXES_MG2.OVERRIDE_FINAL := 7;
   END_IF;
   IF "M_ONE" AND ("DB7224_HMI_AXES".NC_AXES_MG2.OVERRIDE_AUX = 3) THEN
       "DB7224_HMI_AXES".NC_AXES_MG2.OVERRIDE_FINAL := 15;
   END_IF;
   IF "M_ONE" AND ("DB7224_HMI_AXES".NC_AXES_MG2.OVERRIDE_AUX = 4) THEN
       "DB7224_HMI_AXES".NC_AXES_MG2.OVERRIDE_FINAL := 9;
   END_IF;
   IF "M_ONE" AND ("DB7224_HMI_AXES".NC_AXES_MG2.OVERRIDE_AUX = 5) THEN
       "DB7224_HMI_AXES".NC_AXES_MG2.OVERRIDE_FINAL := 26;
   END_IF;
END_REGION
END_FUNCTION
